VAR CONSTANT 		
	MAX_SEND_STRING_SIZE									:	INT := 1024;
END_VAR
VAR_OUTPUT CONSTANT
{attribute 'displaymode':='binary'}
	OPTION_SYSLOG_WITH_FACILITY_SEVERITY_CODE				:	BYTE := 2#0000_0001;
{attribute 'displaymode':='binary'}
	OPTION_SYSLOG_WITH_RFC_HEADER							:	BYTE := 2#0000_0010;
{attribute 'displaymode':='binary'}
	OPTION_SYSLOG_WITH_CR									:	BYTE := 2#0000_0100; 
	{attribute 'displaymode':='binary'}
	OPTION_SYSLOG_WITH_LF									:	BYTE := 2#0000_1000; 
{attribute 'displaymode':='binary'}
//	OPTION_SYSLOG_WITH_TCP_MODE								:	BYTE := 2#0001_0000;
{attribute 'displaymode':='binary'}
	OPTION_SEND_STORED_MSG_WITH_DISABLE						: 	BYTE := 2#0010_0000; //Send stored messages if FB gets disabled to clear buffer
{attribute 'displaymode':='binary'}
	OPTION_ENABLE_BUFFER_ERROR								: 	BYTE := 2#0100_0000; //The FB changes to error state if the buffer was not emptied in time 	
{attribute 'displaymode':='binary'}
	OPTION_ENABLE_DEBUG										:	BYTE := 2#1000_0000; //Creates ADS log entries for conection events and errors
END_VAR
VAR_INPUT
	Enable													: 	BOOL;	//Enables sending new messages
	ResetTrig												:	BOOL;	//Ack error message
{attribute 'displaymode':='binary'}
	Options													:	BYTE := OPTION_SYSLOG_WITH_FACILITY_SEVERITY_CODE ; //option constants are alreay predefined, so they can accordingly be passed symbolically to the block
	SizeOfBuffer											:	UDINT := 2560; //Size of memory allocated from ads router memory pool by DoubleBuffer instance
	LocalHost	 											: 	T_IPv4Addr;  	//Local (client) address. String containing an (Ipv4) Internet Protocol dotted address. 
	LocalPort												:	UDINT := 515;	//Local (client) Internet Protocol (IP) port. (TCP Port = 1468) *)	
	RemoteHost	 											: 	T_IPv4Addr;  	//Remote (server) address. String containing an (Ipv4) Internet Protocol dotted address. 
	RemotePort												:	UDINT := 514;	//Remote (server) Internet Protocol (IP) port. (TCP Port = 1468) 
	Facility												:	BYTE := 16; 	//Default local 16
	Severity 												:	BYTE := 7; 		//0=Emergency/1=Alert/2=Critical/3=Error/4=Warning/5=Notice/6=Informational/7=Debug
	Tag														:	STRING(32) := ''; //Process name or local host by default
	LogPriorityLevel										:	UINT := 0; 		//Correlate to EventClass prioritys - see Para.EVENT_HANDLING_CONFIG prioritys
END_VAR                 				
VAR_OUTPUT              				        			
	Online													:	BOOL;		//TRUE if coonection is sucessful etablished
	hSocket													: 	T_HSOCKET ; //UDP Socket handle
	CntNoOfStoredMsgs										:	INT;
	TimeSendMsgs											:	TIME;
	Busy													: 	BOOL;  //Sending busy
	Error													: 	BOOL;	//Error occured
{attribute 'displaymode':='hex'}
	ErrorId													:	UDINT;	//See Beckhoff TF6310/ADS documentation for more information regarding error code
	ErrorFnc												:	STRING(20); //Error source 
	WinsockErrorId											:	E_WinsockError; //Winsocket error enum - see TF6310 documentation for further information
END_VAR
VAR
(* Memory ************************************************************)
	State													: 	INT := 0;
	StartTimeSendMsgs										:	TIME;
	SendErrorCnt											:	UINT;
	HeaderString											:	STRING;
	SendString												:	STRING(MAX_SEND_STRING_SIZE);
	SendStringLen											:	INT;
	_Severity												:	BYTE;
	LastMessageData											: 	LogbookData;
	LastEventClass											:	E_TcEventClass := TC2_SYSTEM.TCEVENTCLASS_NONE;
	
(* Trigger *****************************************************************)

(* Timer ******************************************************************)

(* Blocks ***************************************************************)
	DblBuffer												:	DoubleBuffer;
	SocketClose												:	FB_SocketClose := (tTimeout := DEFAULT_ADS_TIMEOUT);
	SocketUdpCreate 										:	FB_SocketUdpCreate := (tTimeout := DEFAULT_ADS_TIMEOUT);
	SocketUdpSend											:	FB_SocketUdpSendTo := (tTimeout := T#10S);

(* Dummys *******************************************************************)
	i,j														:	INT;
END_VAR
(* 
Facality Description:
00 Kernel message
01 user-level messages
02 mail system
03 system daemons
04 security/authorization messages
05 messages generated internally by syslogd
06 line printer subsystem
07 network news subsystem
08 UUCP subsystem
09 clock daemon
10 security/authorization messages
11 FTP daemon
12 NTP subsystem
13 log audit
14 log alert
15 clock daemon
16 local10
17 local11
18 local12
19 local13
20 local14
21 local15
22 local16
23 local17

Severity Description:
0 Emergency
1 Alert
2 Critical
3 Error
4 Warning
5 Notice
6 Informational
7 Debug
*)

(* Logbook subscriber to send sys log messages via UDP 				*)
(********************************************************************)

(* Server connection ************************************************)
	CASE state OF
	0:
		IF Error
		THEN
			IF NOT Enable OR ResetTrig 
			THEN //Reset error
				Error										:= FALSE;
				ErrorId										:= 0;
				ErrorFnc									:= '';	
				WinsockErrorId								:= WSOK;			
			END_IF		
		ELSIF Online
		THEN
			IF DblBuffer.ReadyToRead 			
			THEN
				CntNoOfStoredMsgs							:= 0;
				StartTimeSendMsgs							:= TIME();

				SocketUdpSend(
					sSrvNetId	:= , 
					hSocket		:= hSocket, 
					sRemoteHost	:= RemoteHost, 
					nRemotePort	:= RemotePort, 
					cbLen		:= DblBuffer.SizeOfDataToRead, 
					pSrc		:= DblBuffer.pDataToRead, 
					bExecute	:= TRUE, 
					tTimeout	:= , 
					bBusy		=> , 
					bError		=> , 
					nErrId		=> );
													
				state										:= 20;
			END_IF
		ELSIF Enable			
		THEN
			DblBuffer.SizeOfMemory							:= SizeOfBuffer;
			SocketUdpCreate(bExecute := FALSE);
			SocketClose(bExecute := FALSE);
			SocketUdpSend(bExecute := FALSE);
			Online											:= FALSE;
			Busy											:= TRUE;
			Error											:= FALSE;
			ErrorId											:= 0;
			ErrorFnc										:= '';	
			WinsockErrorId									:= WSOK;
			
			IF NOT SocketUdpCreate.bBusy
				AND NOT SocketClose.bBusy
				AND NOT SocketUdpSend.bBusy
			THEN
				state										:= 10;
			END_IF	
		ELSE //Disabled
			IF NOT DblBuffer.Empty AND Options.5
			THEN //Write rest of buffer
				IF NOT DblBuffer.ReadyToRead THEN DblBuffer.setReadyToRead(TRUE); END_IF 
				CntNoOfStoredMsgs							:= 0;
				StartTimeSendMsgs							:= TIME();
				SocketUdpSend(
					sSrvNetId	:= , 
					hSocket		:= hSocket, 
					sRemoteHost	:= RemoteHost, 
					nRemotePort	:= RemotePort, 
					cbLen		:= DblBuffer.SizeOfDataToRead, 
					pSrc		:= DblBuffer.pDataToRead, 
					bExecute	:= TRUE, 
					tTimeout	:= , 
					bBusy		=> , 
					bError		=> , 
					nErrId		=> );
				State										:= 20;
			ELSE //Close socket
				State										:= 30;
			END_IF			
		END_IF

	(* Create Socket *******************************************************)
	10: 
		SocketUdpCreate(
			sSrvNetId	:= , 
			sLocalHost	:= LocalHost, 
			nLocalPort	:= LocalPort, 
			bExecute	:= TRUE, 
			tTimeout	:= , 
			bBusy		=> , 
			bError		=> , 
			nErrId		=> , 
			hSocket		=> hSocket);
			
		IF NOT SocketUdpCreate.bBusy
		THEN
			IF SocketUdpCreate.bError
			THEN
				Error										:= TRUE;
				ErrorId										:= SocketUdpCreate.nErrId;
				ErrorFnc									:= 'SocketUdpCreate';
				WinsockErrorId								:= ADSERROR_TO_WSERROR(ErrorId);
				
				IF (Options AND OPTION_ENABLE_DEBUG) = 1
				THEN
					AdsLogError(CONCAT('LogbookClientSysLog | SocketUdpCreate %s | error id 16#', DWORD_TO_HEXSTR(TO_DWORD(ErrorID),4,FALSE)) ,HSOCKET_TO_STRING(SocketUdpCreate.hSocket));
				END_IF	

				state										:= 30;
			ELSE				
				hSocket.remoteAddr.sAddr					:= RemoteHost;
				hSocket.remoteAddr.nPort					:= RemotePort;
				
				IF (Options AND OPTION_ENABLE_DEBUG) = 1
				THEN
					AdsLogError(CONCAT('LogbookClientSysLog | SocketUdpCreate %s done', '') , HSOCKET_TO_STRING(SocketUdpCreate.hSocket));
				END_IF	
				
				Online 										:= TRUE;
				state										:= 0;
			END_IF		
			SocketUdpCreate(bExecute:= FALSE);
		END_IF		
		
	(* Send message ****************************************************)
	20:
		SocketUdpSend(
			sSrvNetId	:= , 
			hSocket		:= hSocket, 
			sRemoteHost	:= RemoteHost, 
			nRemotePort	:= RemotePort, 
			cbLen		:= DblBuffer.SizeOfDataToRead, 
			pSrc		:= DblBuffer.pDataToRead, 
			bExecute	:= TRUE, 
			tTimeout	:= , 
			bBusy		=> , 
			bError		=> , 
			nErrId		=> );
					
		IF NOT SocketUdpSend.bBusy
		THEN
			IF SocketUdpSend.bError
			THEN
				IF SendErrorCnt >= 3
				THEN
					Error									:= TRUE;
					ErrorId									:= SocketUdpSend.nErrId;
					ErrorFnc								:= 'SocketUdpSend';
					WinsockErrorId							:= ADSERROR_TO_WSERROR(ErrorId);
	
					IF (Options AND OPTION_ENABLE_DEBUG) = 1
					THEN
						AdsLogError(CONCAT('LogbookClientSysLog | SocketUdpSend %s | error id 16#', DWORD_TO_HEXSTR(TO_DWORD(ErrorID),4,FALSE)) ,HSOCKET_TO_STRING(SocketUdpCreate.hSocket));
					END_IF	
					
					State									:= 30; //Close socket
				ELSE //Try to send a second time
					SendErrorCnt							:= SendErrorCnt + 1;
				END_IF
			ELSE				
				SendErrorCnt								:= 0;	
				State										:= 0;			
			END_IF 
			DblBuffer.setReadyToRead(FALSE);
			SocketUdpSend(bExecute := FALSE);
		END_IF
		
	(* Close socket ***********************************************)
	30:	
		SocketClose(
			sSrvNetId	:= , 
			hSocket		:= SocketUdpCreate.hSocket, 
			bExecute	:= TRUE, 
			tTimeout	:= , 
			bBusy		=> , 
			bError		=> , 
			nErrId		=> );

		IF NOT SocketClose.bBusy
		THEN
			Online											:= FALSE;
			IF SocketClose.bError 
				AND NOT Error
			THEN
				Error										:= TRUE;
				ErrorId										:= SocketClose.nErrId;
				ErrorFnc									:= 'SocketUdpClose';
				WinsockErrorId								:= ADSERROR_TO_WSERROR(ErrorId);
				
				IF (Options AND OPTION_ENABLE_DEBUG) = 1
				THEN
					AdsLogError( CONCAT('LogbookClientSysLog | SocketClose %s | error id 16#', DWORD_TO_HEXSTR(TO_DWORD(ErrorID),4,FALSE)) ,HSOCKET_TO_STRING(SocketClose.hSocket));
				END_IF

				state										:= 0;				
			ELSE    
				IF (Options AND OPTION_ENABLE_DEBUG) = 1
				THEN
					AdsLogError( CONCAT('LogbookClientSysLog | SocketClose %s done', '') , HSOCKET_TO_STRING(SocketClose.hSocket));
				END_IF	
                                        
				state										:= 0;
			END_IF		
			SocketClose(bExecute := FALSE);
		END_IF		
			
	END_CASE
	
(* Status *****************************************************************)
	Busy 													:= State <> 0;
	
(**************************************************************************)

METHOD PUBLIC FINAL addNewMessage : BOOL //Return value = TRUE if execution successful finished
VAR_IN_OUT
	data													:	LogbookData;
END_VAR
	IF Enable AND NOT Error
	THEN	
		LastMessageData									:= Data;
		LastEventClass.0								:= LastMessageData.Options.8;
		LastEventClass.1								:= LastMessageData.Options.9;
		LastEventClass.2								:= LastMessageData.Options.10;
		LastEventClass.3								:= LastMessageData.Options.11;
		
		CASE LastEventClass OF
		TC2_SYSTEM.TCEVENTCLASS_NONE		: _Severity		:= Severity; 		
		TC2_SYSTEM.TCEVENTCLASS_MESSAGE		: _Severity		:= 4;				
		TC2_SYSTEM.TCEVENTCLASS_HINT		: _Severity		:= 5;				
		TC2_SYSTEM.TCEVENTCLASS_STATEINFO	: _Severity		:= 6;				
		TC2_SYSTEM.TCEVENTCLASS_INSTRUCTION	: _Severity		:= 6;			 											
		TC2_SYSTEM.TCEVENTCLASS_WARNING		: _Severity		:= 4;	 			
		TC2_SYSTEM.TCEVENTCLASS_MAINTENANCE	: _Severity		:= 1;	 				 														
		TC2_SYSTEM.TCEVENTCLASS_ALARM		: _Severity		:= 0;	 			
		TC2_SYSTEM.TCEVENTCLASS_PARAMERROR	: _Severity		:= 3;	 			
		ELSE                                                                                     
			_Severity									:= 7;				
		END_CASE
	
		IF (LogPriorityLevel = 0 OR_ELSE GetEventClassPriority(LastEventClass) > LogPriorityLevel)
			AND_THEN CreateMsg(LastMessageData.Msg,LastMessageData.Timestamp ,_Severity)
		THEN
			IF DblBuffer.addData(ADR(SendString),TO_UDINT(SendStringLen)) <> S_OK
				AND Options.6
			THEN
				Error										:= TRUE;
				ErrorId										:= HRESULT_TO_ADSERROR(DblBuffer.hr);	
			ELSE
				CntNoOfStoredMsgs							:= CntNoOfStoredMsgs + 1;
			END_IF
		END_IF
		
		addNewMessage										:= NOT Error;	
	ELSE
		addNewMessage										:= FALSE;	
	END_IF
END_METHOD

METHOD PRIVATE FINAL createMsg : BOOL
VAR_IN_OUT
	MsgTxt													:	T_MaxString; (* 80/255 Zeichen *)
	MsgTime													:	TIMESTRUCT;	
	Severity												:	BYTE;
END_VAR                 									
VAR                     									
	TimeStamp												:	STRING(20);
	LenTxt													:	UDINT;
	LenHeader												:	UDINT;
END_VAR
	//Create Syslog msg
	IF (Options AND OPTION_SYSLOG_WITH_FACILITY_SEVERITY_CODE) <> 0 
	THEN 
		HeaderString 										:= REPLACE('<P>',BYTE_TO_STRING(SHL(FACILITY,3) OR (Severity AND BYTE#0000_0111)),1,2);
		             										
	ELSE             										
		HeaderString 										:= '';
	END_IF
	
	IF (Options AND OPTION_SYSLOG_WITH_RFC_HEADER) <> 0 
	THEN 
		//Sep 10 08:31:10
		CASE MsgTime.wMonth OF
		1: HeaderString 									:= CONCAT(HeaderString, ' Jan ');
		2: HeaderString 									:= CONCAT(HeaderString, ' Feb ');
		3: HeaderString 									:= CONCAT(HeaderString, ' Mar ');
		4: HeaderString 									:= CONCAT(HeaderString, ' Apr ');
		5: HeaderString 									:= CONCAT(HeaderString, ' May ');
		6: HeaderString 									:= CONCAT(HeaderString, ' Jun ');
		7: HeaderString 									:= CONCAT(HeaderString, ' Jul ');
		8: HeaderString 									:= CONCAT(HeaderString, ' Aug ');
		9: HeaderString 									:= CONCAT(HeaderString, ' Seb ');
		10:HeaderString 									:= CONCAT(HeaderString, ' Oct ');
		11:HeaderString 									:= CONCAT(HeaderString, ' Nov ');
		12:HeaderString 									:= CONCAT(HeaderString, ' Dec ');
		END_CASE
			
		HeaderString 										:= CONCAT(HeaderString,WORD_TO_STRING(MsgTime.wDay));
		HeaderString 										:= CONCAT(HeaderString, ' ');
					
		IF MsgTime.wHour <10 
		THEN
			TimeStamp 										:= CONCAT(' 0',WORD_TO_STRING(MsgTime.wHour));
		ELSE
			TimeStamp 										:= WORD_TO_STRING(MsgTime.wHour);
		END_IF
		
		TimeStamp 											:= CONCAT(TimeStamp,':');
		
		IF MsgTime.wMinute < 10 
		THEN
			TimeStamp 										:= CONCAT(TimeStamp,CONCAT('0',WORD_TO_STRING(MsgTime.wMinute)));
		ELSE          										
			TimeStamp 										:= CONCAT(TimeStamp,WORD_TO_STRING(MsgTime.wMinute));
		END_IF
		
		TimeStamp 											:= CONCAT(TimeStamp,':');
		
		IF MsgTime.wSecond < 10 
		THEN
			TimeStamp 										:= CONCAT(TimeStamp,CONCAT('0',WORD_TO_STRING(MsgTime.wSecond)));
		ELSE
			TimeStamp 										:= CONCAT(TimeStamp,WORD_TO_STRING(MsgTime.wSecond));
		END_IF
		HeaderString 										:= CONCAT(HeaderString,TimeStamp);
		HeaderString 										:= CONCAT(HeaderString,' ');
					
		(* ' sourcename eintragen (IP) *)
		HeaderString 										:= CONCAT(HeaderString, hSocket.localAddr.sAddr ); 
		HeaderString 										:= CONCAT(HeaderString,' '); 
		
		(* Tag *)
		IF Len(Tag) > 0
		THEN
			HeaderString									:= CONCAT(HeaderString,Tag);
			HeaderString 									:= CONCAT(HeaderString,' '); 
		END_IF
	END_IF
	
	IF Options.2 
	THEN //CR
		MsgTxt												:= CONCAT(MsgTxt,'$r');
	END_IF
	
	IF Options.3 
	THEN //LF
		MsgTxt												:= CONCAT(MsgTxt,'$n');
	END_IF
	
	(* Msg *)
	SendString												:= HeaderString;
	SendStringLen											:= MIN(MAX_SEND_STRING_SIZE,(LEN(HeaderString) + Len(MsgTxt)));
	MEMCPY(ADR(SendString) + LEN(HeaderString), ADR(MsgTxt) , INT_TO_UDINT(LEn(MsgTxt)));
	SendString[SendStringLen] 								:= 0; //Terminate string
	
	CreateMsg												:= TRUE;
END_METHOD

PROPERTY PUBLIC optAdd_CR : BOOL
GET
optAdd_CR := Options.2;
END_GET
SET
OPtions.2 := optAdd_CR;
END_SET
END_PROPERTY

PROPERTY PUBLIC optAdd_LF : BOOL
GET
optAdd_LF := Options.3;
END_GET
SET
Options.3 := optAdd_LF;
END_SET
END_PROPERTY

PROPERTY PUBLIC optEnabelDebugMode : BOOL
GET
optEnabelDebugMode := Options.7;
END_GET
SET
Options.7 := optEnabelDebugMode;
END_SET
END_PROPERTY

PROPERTY PUBLIC optEnableBufferError : BOOL
GET
optEnableBufferError := Options.6;
END_GET
SET
OPtions.6				:= optEnableBufferError;
END_SET
END_PROPERTY

PROPERTY PUBLIC optEnableFacilitySeverityCode : BOOL
GET
 optEnableFacilitySeverityCode := Options.0;
END_GET
SET
Options.0 := optEnableFacilitySeverityCode;
END_SET
END_PROPERTY

PROPERTY PUBLIC optEnableRFCHeader : BOOL
GET
optEnableRFCHeader := Options.1;
END_GET
SET
Options.1 := optEnableRFCHeader;
END_SET
END_PROPERTY

PROPERTY PUBLIC optSendMsgIfDisabled : BOOL
GET
optSendMsgIfDisabled := Options.5;
END_GET
SET
Options.5 := optSendMsgIfDisabled;
END_SET
END_PROPERTY

{attribute 'monitoring' := 'call'}
PROPERTY PUBLIC isBusy : BOOL
GET
isBusy											:= DblBuffer.Full and Enable and not Error and DblBuffer.fillLevel >= MAX_BUFFER_LEVEL;
END_GET
END_PROPERTY

END_FUNCTION_BLOCK

// POUs/Logging/LogbookSubWriteFile
{attribute 'no_check' := ''}
//The LogbooSubWriteFile writes log entries handover by the LogbookPuplisher into txt files
//The files could be stored or overwritten on a daily (Today/Yesterday), weekly (1-7 days) or monthly base (1-31 days) - see DeleteMode Parameter  
{attribute 'enable_dynamic_creation'}
FUNCTION_BLOCK LogbookSubWriteFile IMPLEMENTS I_LogbookSubscriber
VAR CONSTANT
	MAX_BUFFER_LEVEL										:	INT := 85; //If buffer fill level reaches 85% Fb will appear as "busy2 to the LogBookPuplisher 
END_VAR
VAR_OUTPUT CONSTANT 
	STRING_LINE_END_SIGN									: STRING(6) := PARAM.LOGBOOK_SUB_WRT_FILE_LINE_END_SIGN; //e.g. $n
	DELAY_CLOSE_FILE										: TIME := PARAM.LOGBOOK_SUB_WRT_FILE_DELAY_FILE_CLOSE;  //see library parameter to customize parameter	
		
	DELETE_MODE_DAILY										: INT := 0; //FB will write a file with <Filename>_TODAY and rename existing file to <Filename>_YESTERDAY on a new day
	DELETE_MODE_WEEKLY										: INT := 1; //FB will create a file for each day of week <Filenme>_DAY_1..7
	DELETE_MODE_MONTHLY										: INT := 2; //FB will create a file for each day of month <Filenme>_DAY_n (n=1..31) 
	DELETE_MODE_DISABLED									: INT := 3; //FB will write an endless file, see options .7 to start with an empty file on a new day  

	{attribute 'displaymode':='binary'}
	OPTION_ADD_TIMESTAMP_TO_MSG								: BYTE := 2#0000_0001; //Add message time to file entry - see next option for date option
	{attribute 'displaymode':='binary'}
	OPTION_ADD_DATE_TO_TIMESTAMP							: BYTE := 2#0000_0010; //Only active if option "OPTION_ADD_TIMESTAMP_TO_MSG" is set 
	{attribute 'displaymode':='binary'}
	OPTION_ADD_CLASS_TO_MSG									: BYTE := 2#0000_0100; //Event class text will be added to entries
	{attribute 'displaymode':='binary'}
	OPTION_ENABLE_BUFFER_ERROR								: BYTE := 2#0100_0000; //The FB changes to error state if the buffer was not emptied in time 
	{attribute 'displaymode':='binary'}
	OPTION_START_WITH_NEW_FILE								: BYTE := 2#1000_0000; //Create empty file with enable flag instead open and continie existing file
END_VAR                     								
VAR_INPUT                   								
	Enable													: BOOL; //Enable write log entries to file
	ResetTrig												: BOOL; //Reset internal error 
{attribute 'displaymode':='binary'}
	Options													: BYTE := 2#00000000; // Bit 0 = Add msg timestamp to entry string 	
	DeleteMode												: INT(DELETE_MODE_DAILY..DELETE_MODE_DISABLED) := DELETE_MODE_DAILY;
	Path													: STRING := 'C:\temp'; //Path and filename
	Filetype												: STRING(6) := '.log'; //file tpye
	LoggedDay												: WORD;	//Init for logged day of month to avoid new and empty log file after reboot.
	SizeOfBuffer											: UDINT := 2560; //Size of memory allocated from router pool to accumulate messages until they get written to the file (0=Write message immediately)
END_VAR                     								
VAR_IN_OUT                  								
	SystemTime												: TIMESTRUCT; //System time
END_VAR                     								
VAR_OUTPUT       
	CntNoOfStoredMsgs										: INT; //No of messages added to buffer 

	hFile													: UINT;  
	Busy													: BOOL; //Write msg to file active   
	Error													: BOOL;        			
{attribute 'displaymode':='hex'}					
	ErrorId													: UDINT; //Ads error Id of file handling function blocks
END_VAR                     								
VAR            
//local ************************************************************************************
	State													: INT := 0;
	LastLoggedDay											: WORD;
	Rebooted												: BOOL;
	LastMessageData											: LogbookData;
	StartTimeWriteData										: TIME;	
	TimeWriteFile											: TIME; 
	MemMessage												: U_MAX_STRING;
	MemLenStrEndLine										: INT;	
	MemStartOfEndLine										: DINT;	
	MemPath													: STRING;
	
//trigger *********************************************************************************

//timer ***********************************************************************************
	tonCloseFile											:	ton;

//instances ***********************************************************************************     
	DblBuffer												: DoubleBuffer;        								
	FILEOPEN												: FB_FileOpen := (sNetId:='',tTimeout:=DEFAULT_ADS_TIMEOUT, ePath:=PATH_GENERIC);
	FILECLOSE												: FB_FileClose := (sNetId:='',tTimeout:=DEFAULT_ADS_TIMEOUT);
	FILEWRITE												: FB_FileWrite := (sNetId:='',tTimeout:=DEFAULT_ADS_TIMEOUT);
	FILEDELETE												: FB_FileDelete := (sNetId:='',tTimeout:=DEFAULT_ADS_TIMEOUT);
	FILERENAME												: FB_FileRename := (sNetId:='',tTimeout:=DEFAULT_ADS_TIMEOUT, ePath:=PATH_GENERIC);

//Dummys ****************************************************************************************
	i,j,n													: INT;
	_UINT													:	UINT;
END_VAR

	(* Logbook subscriber write messages to file			*)
	(********************************************************)

(* Sequence started by method "NewMessage" or a new day ***************************************************)
	CASE State OF
	0:	
		IF Error
		THEN
			IF ResetTrig OR NOT Enable
			THEN
				Error										:= FALSE;
				ErrorId										:= 0;
				FileOpen(bExecute:=FALSE);
				FileClose(bExecute:=FALSE);
				FileDelete(bExecute:=FALSE);
				FileRename(bExecute:=FALSE);
				FileWrite(bExecute:=FALSE);
			END_IF
		ELSIF Enable
		THEN
			IF SystemTime.wDay = 0
			THEN
				Error										:= TRUE;
				ErrorId										:= E_AdsErr.DEVICE_INVALIDPARM; //Systemtime invalid 				
			ELSIF hFile = 0 // close last before opening next file
				AND(LastLoggedDay <> SystemTime.wDay OR MemPath <> Path) 			
			THEN //create new or overwrite existing file if new day begins
				DblBuffer.SizeOfMemory						:= SizeOfBuffer;
						
				MemLenStrEndLine							:= LEN(STRING_LINE_END_SIGN);
				MemStartOfEndLine							:= TO_DINT(LIMIT(1,PARAM.LOGBOOK_MAX_MSG_STRING_LENGHT - TO_UDINT(MemLenStrEndLine) + 1, PARAM.LOGBOOK_MAX_MSG_STRING_LENGHT - 1));
				Rebooted									:= LastLoggedDay = 0;
 	
				(* Init last logged day of month and path on startup *)
				IF Rebooted 
				THEN 
					MemPath  								:= Path;
					LastLoggedDay 							:= SEL(LoggedDay > 0, 0, LoggedDay); 
				END_IF	
				
				CASE DeleteMode OF
				DELETE_MODE_WEEKLY: //Day 1 to 7
					FileOpen.sPathName 						:= CONCAT(Path, CONCAT('_DAY_',WORD_TO_STRING(SystemTime.wDayOfWeek)));
					CASE SystemTime.wDayOfWeek OF
					0:FileOpen.sPathName 					:= CONCAT(FileOpen.sPathName,'_SUN' );
					1:FileOpen.sPathName 					:= CONCAT(FileOpen.sPathName,'_MON' );
					2:FileOpen.sPathName					:= CONCAT(FileOpen.sPathName,'_TUE' );
					3:FileOpen.sPathName 					:= CONCAT(FileOpen.sPathName,'_WED' );
					4:FileOpen.sPathName 					:= CONCAT(FileOpen.sPathName,'_THU' );
					5:FileOpen.sPathName 					:= CONCAT(FileOpen.sPathName,'_FRI' );
					6:FileOpen.sPathName 					:= CONCAT(FileOpen.sPathName,'_SAT' );
					ELSE
						FileOpen.sPathName 					:= CONCAT(FileOpen.sPathName,'_UNKNOW' );
					END_CASE
					
				DELETE_MODE_MONTHLY: //Every Month - Day 1-n
					FileOpen.sPathName 						:= CONCAT(Path, CONCAT('_',WORD_TO_STRING(SystemTime.wDay)));
					
				DELETE_MODE_DISABLED:		
					FileOpen.sPathName			 			:= Path;
					
				ELSE //DELETE_MODE_DAILY as default
					FileOpen.sPathName 						:= CONCAT(Path, '_TODAY');	//Today and yesterday
				
				END_CASE
				FileOpen.sPathName							:= CONCAT(FileOpen.sPathName,Filetype);
									
				IF DeleteMode <> DELETE_MODE_DISABLED AND LastLoggedDay <> SystemTime.wDay 
				THEN //New day - start with new file	
					FileOpen(bExecute:=FALSE,nMode := FOPEN_MODEWRITE OR FOPEN_MODETEXT OR FOPEN_MODEPLUS);							
					IF DeleteMode = DELETE_MODE_DAILY
					THEN //Rename old file first		
						FILERENAME(bExecute:=FALSE, sOldName := FileOpen.sPathName, sNewName := CONCAT(Path, CONCAT('_YESTERDAY',Filetype)));
						FILEDELETE(bExecute:=FALSE, sPathName := FILERENAME.sNewName );
						FileClose(bExecute:=hFile <> 0 , hFile := hFile);
						state								:= 10;
					ELSE //Create new file directly
						FileOpen(bExecute:=TRUE,nMode := FOPEN_MODEWRITE OR FOPEN_MODETEXT OR FOPEN_MODEPLUS);
						state								:= 1;
					END_IF
				ELSE //write endless file with given name and open existing one if selected 														
					FileOpen(bExecute:= TRUE , nMode:=SEL(Options.7 ,FOPEN_MODEAPPEND,FOPEN_MODEWRITE) OR FOPEN_MODETEXT OR FOPEN_MODEPLUS );
					state									:= 1;
				END_IF	 	
	
				(* Record current day of detected new beginning day *)
				LastLoggedDay 								:= SystemTime.wDay;	
				MemPath  									:= Path;
				
			ELSE
				tonCloseFile(IN := NOT DblBuffer.Empty ,PT := DELAY_CLOSE_FILE); 
				IF DblBuffer.ReadyToRead
					OR tonCloseFile.Q
				THEN
					IF NOT DblBuffer.ReadyToRead THEN DblBuffer.setReadyToRead(TRUE); END_IF 
					FILEWRITE.pWriteBuff 					:= DblBuffer.pDataToRead;
					FILEWRITE.cbWriteLen 					:= DblBuffer.SizeOfDataToRead;
					FILEWRITE.bExecute						:= DblBuffer.SizeOfDataToRead > 0; //Set Write file as marker

					FileClose.bExecute						:= SystemTime.wDay > 0
																AND(LastLoggedDay <> SystemTime.wDay OR MemPath <> Path)
																AND hFile <> 0
																OR tonCloseFile.Q; //Set close file as marker
																
					tonCloseFile(IN := FALSE); //Reset timer....
					CntNoOfStoredMsgs						:= 0;
					StartTimeWriteData						:= TIME();
					
					IF hFile = 0
					THEN
						FileOpen(bExecute:= TRUE , nMode:=SEL(Options.7 ,FOPEN_MODEAPPEND,FOPEN_MODEWRITE) OR FOPEN_MODETEXT OR FOPEN_MODEPLUS ); //Reopen file first
						State								:= 1;
					ELSE
						FILEWRITE(hFile := hFile); //Start write file for efficiency 		
						State								:= 2;
					END_IF					
				END_IF			
			END_IF
						
		ELSE //Not enabled
			IF NOT DblBuffer.Empty
			THEN //Write rest of buffer
				IF NOT DblBuffer.ReadyToRead THEN DblBuffer.setReadyToRead(TRUE); END_IF 
				FILEWRITE(bExecute:=TRUE,hFile:= hFile , pWriteBuff := DblBuffer.pDataToRead, cbWriteLen := DblBuffer.SizeOfDataToRead);	
				CntNoOfStoredMsgs							:= 0;
				StartTimeWriteData							:= TIME();
				FileClose.bExecute							:= TRUE;  //Close file after writing
				State										:= SEL(hFile <> 0 , 1, 2) ; //Open file if not opened
			ELSIF hFile <> 0
			THEN
				FileClose(bExecute:=TRUE , hFile := hFile);
				state										:= 3;	
			END_IF
        END_IF
     
	(* Open file *******************************************************************************)                                          	
	1:                       	
		FileOpen();                                     	
		IF NOT FileOpen.bBusy                           	
		THEN                                            	
			IF FileOpen.bError                          	
			THEN            
				Error										:= TRUE;                            	
				ErrorId										:= FileOpen.nErrId;
				State										:= 0;
			ELSE                                     	
				hFile										:= FileOpen.hFile;       	
				State										:= SEL(FILEWRITE.bExecute, 0, 2) ;
			END_IF
			FileOpen(bExecute:=FALSE);			
		END_IF

	(* Write data to file **********************************************************************)
	2: 
		FILEWRITE(hFile:= hFile);	
		IF NOT FILEWRITE.bBusy
		THEN
			
			IF FILEWRITE.bError
			THEN
				Error										:= TRUE;       
				ErrorId										:= FILEWRITE.nErrId;
				state										:= 0;
			ELSE  
				State										:= SEL(FileClose.bExecute, 0, 3);	
			END_IF		
			TimeWriteFile									:= TIME() - StartTimeWriteData;		
			DblBuffer.setReadyToRead(FALSE);	
			FILEWRITE(bExecute:=FALSE);   	
		END_IF

	(* Close File ******************************************************************************)
	3: 
		FileClose(hFile:= hFile);
		IF NOT FileClose.bBusy
		THEN
			IF FileClose.bError
			THEN
				Error										:= TRUE;       
				ErrorId										:= FileClose.nErrId;
				State										:= 0;
			ELSE                                        	
				hFile										:= 0;
				State										:= 0;
			END_IF
			FileClose(bExecute:=FALSE);
		END_IF

	(* Delete old file and rename exisiting file ********************************************************) 
	10: 
		FileClose();
		FileDelete(bExecute:=NOT FileClose.bBusy);
		IF NOT FileDelete.bBusy AND NOT FileClose.bBusy
		THEN
			IF FileDelete.bError
			THEN //No issue, maybe file is not existing
			//	Error										:= TRUE;       
			//	ErrorId										:= FileDelete.nErrId;
				State										:= 11;
			ELSIF FileClose.bError
			THEN
			//	Error										:= TRUE;       
			//	ErrorId										:= FileClose.nErrId;
				State										:= 11;			
			ELSE                                        	
				State										:= 11;
			END_IF
			FileDelete(bExecute:=FALSE); FileClose(bExecute:=FALSE);
		END_IF
		
	11: //Rename last file to create a new and empty file for today
		FILERENAME(bExecute:=TRUE);
		IF NOT FILERENAME.bBusy
		THEN
			IF FILERENAME.bError
			THEN //No issue, maybe file does not exist
			//	Error										:= TRUE;       
			//	ErrorId										:= FILERENAME.nErrId;
				State										:= 1;
			ELSE                                        	
				State										:= 1;
			END_IF
			FILERENAME(bExecute:=FALSE);	
			FileOpen(bExecute:= TRUE); //Start create new file for today										
		END_IF		
	ELSE
		;
	END_CASE

(* Ack ErrorIds **********************************************************)
	Busy 													:= State <> 0;
(**************************************************************************)

METHOD PUBLIC FINAL addNewMessage : BOOL //Return value = TRUE if execution successful finished
VAR_IN_OUT
	data													:	LogbookData;
END_VAR
	IF Enable AND NOT Error
	THEN		
		CntNoOfStoredMsgs								:= CntNoOfStoredMsgs + 1;
		LastMessageData									:= Data;

		MEMSET(ADR(MemMessage),0,SIZEOF(MemMessage));
		IF Options.0 AND Options.1 //Add date and time to text
		THEN
			MemMessage.text								:=	SYSTEMTIME_TO_STRING(LastMessageData.Timestamp);						
			MemMessage.text 							:=	CONCAT(MemMessage.text, ';');

		ELSIF Options.0 //Add only msg timestamp to text		
		THEN
			MemMessage.text								:=	SYSTEMTIME_TO_STRING(LastMessageData.Timestamp);
			MemMessage.text								:=	MID(MemMessage.text, 12 , 12); //Cut out time
			MemMessage.text 							:=	CONCAT(MemMessage.text, ';');
		END_IF      

		IF Options.2 //Add class of message to text
		THEN
			_UINT.0 									:= LastMessageData.Options.8;
			_UINT.1 									:= LastMessageData.Options.9;
			_UINT.2 									:= LastMessageData.Options.10;
			_UINT.3 									:= LastMessageData.Options.11;		
			MemMessage.text								:= CONCAT(MemMessage.text, GetEventClassText(_UINT));	
			MemMessage.text 							:= CONCAT(MemMessage.text, ';');			
		END_IF
	
		MemMessage.text 								:= CONCAT(MemMessage.text, LastMessageData.Msg);

		IF LEN(MemMessage.text) < MemStartOfEndLine
		THEN //Still enough space for end line signs
			MemMessage.text 							:= CONCAT(MemMessage.text,STRING_LINE_END_SIGN );
		ELSE //Overwrite last chars with endline signs
			MEMCPY(ADR(MemMessage.text[MemStartOfEndLine]),ADR(STRING_LINE_END_SIGN),TO_UDINT(MemLenStrEndLine));
		END_IF
		
		IF DblBuffer.addString(MemMessage.text) <> S_OK
			AND Options.6
		THEN
			Error										:= TRUE;
			ErrorId										:= HRESULT_TO_ADSERROR(DblBuffer.hr);	
		END_IF
		
		addNewMessage									:= NOT Error;
	ELSE
		addNewMessage									:= FALSE;
	END_IF
END_METHOD

PROPERTY PUBLIC optAddDateToMsg : BOOL
GET
optAddDateToMsg := Options.1;
END_GET
SET
Options.1 := optAddDateToMsg and optAddTimeToMsg;
END_SET
END_PROPERTY

PROPERTY PUBLIC optAddEventClassToMsg : BOOL
GET
optAddEventClassToMsg := Options.2;
END_GET
SET
Options.2 := optAddEventClassToMsg ;
END_SET
END_PROPERTY

PROPERTY PUBLIC optAddTimeToMsg : BOOL
GET
optAddTimeToMsg := Options.0;
END_GET
SET
IF optAddTimeToMsg 
THEN
	Options.0 := TRUE;
ELSE
	Options.0 := Options.1 := FALSE;
END_IF
END_SET
END_PROPERTY

PROPERTY PUBLIC optEnableBufferError : BOOL
GET
optEnableBufferError := Options.6;
END_GET
SET
OPtions.6				:= optEnableBufferError;
END_SET
END_PROPERTY

PROPERTY PUBLIC optSendMsgIfDisabled : BOOL
GET
optSendMsgIfDisabled := Options.5;
END_GET
SET
Options.5 := optSendMsgIfDisabled;
END_SET
END_PROPERTY

PROPERTY PUBLIC optStartNewFile : BOOL
GET
optStartNewFile := Options.7;
END_GET
SET
OPtions.7				:= optStartNewFile;
END_SET
END_PROPERTY

{attribute 'monitoring' := 'call'}
PROPERTY PUBLIC isBusy : BOOL
GET
isBusy											:= DblBuffer.Full and Enable and not Error and DblBuffer.fillLevel >= MAX_BUFFER_LEVEL;
END_GET
END_PROPERTY

END_FUNCTION_BLOCK

// POUs/Motion/TF50xx-NC/00_Base/AxFbBase
//Axis FB template, inherited Execute, Busy etc from FbBase   
FUNCTION_BLOCK AxFbBase EXTENDS FbBase 
VAR_INPUT
	rAxis													: REFERENCE TO AXIS_REF := 0; //Reference to AXIS_REF 
END_VAR
VAR_IN_OUT
END_VAR
VAR_OUTPUT
	Active													: BOOL ; // If the axis movement is controlled by several functions, the Active output of each block indicates that the axis executes the command. 
	CmdAborted												: BOOL ; // TRUE if a command is interrupted through another block (Busy and Error = FALSE)
	ErrorText												: STRING(40); //Error text with name of internal used FB which causes the error
END_VAR
VAR 
	LastErrorId												: UDINT := 0; //Last error id
END_VAR

END_FUNCTION_BLOCK

// POUs/Motion/TF50xx-NC/00_Base/I_AxNcBase
INTERFACE I_AxNcBase EXTENDS __SYSTEM.IQueryInterface

METHOD PUBLIC noAction : BOOL //Return value = TRUE if busy of home and motion 
VAR_INPUT
END_VAR
END_METHOD

{attribute 'monitoring' := 'call'}
PROPERTY rAdmin : REFERENCE TO AxAdmin
GET
END_GET
END_PROPERTY

{attribute 'monitoring' := 'call'}
PROPERTY rAxisRef : REFERENCE TO AXIS_REF
GET
END_GET
END_PROPERTY

{attribute 'monitoring' := 'call'}
PROPERTY rErrHdl : REFERENCE to ERROR_HDL
GET
END_GET
SET
END_SET
END_PROPERTY

METHOD reset : Bool
VAR_INPUT
END_VAR
END_METHOD

{attribute 'monitoring' := 'call'}
PROPERTY rHome : REFERENCE TO AxHoming
GET
END_GET
END_PROPERTY

{attribute 'monitoring' := 'call'}
PROPERTY rPara : REFERENCE TO AxPara
GET
END_GET
END_PROPERTY

END_INTERFACE

// POUs/Motion/TF50xx-NC/01_Main/AxAdmin
{attribute 'no_check'}
//Nc-axis administration - Axis reset, set operation and override
//based on Tc2_MC2 library
//Call cyclic to update AXIS_REF.status
FUNCTION_BLOCK AxAdmin 
VAR_INPUT
	ResetTrig												:	BOOL := FALSE; // Reset NC Error and restart current cmd if possible
	Enable													: 	BOOL := FALSE; // Cyclic NCAxis enable operational - FALSE = Stop 
	EnablePos												: 	BOOL := FALSE; // feed enable positiv 
	EnableNeg												: 	BOOL := FALSE; // feed enable negative 
	BufferMode												:	MC_BufferMode := MC_Aborting;	(* 	MC_Aborting,
																									MC_Buffered,
																									MC_BlendingLow,
																									MC_BlendingPrevious,
																									MC_BlendingNext,
																									MC_BlendingHigh *) 
                                							
	Override												:	LREAL; // Override 
	PT_Ready												:	TIME := T#10MS; //Delay of ready signal after NC-Axis has been enabled
	ShowNCErrIfDisabled										:	BOOL := FALSE; // FB reports and NC-Error even if axis has been diabled
	EnableNcDebugFlag										:	BOOL := FALSE; //TRUE writes every MC2 start command into TwinCAT and Windows logger. 
	ExeMcStopToDisable										:	BOOL := FALSE; //Initiats the execution of MC_Stop on a running axis if "Enable" is set to FALSE
	Dec														:	LREAL := 0.0; //Deceleration during disable, if the value is 0, the deceleration parameterized with the last Move command is used / see also ExeMcStopToDisable
	Jerk													:	LREAL := 0.0; //Jerk during disable, if the value is 0, the deceleration parameterized with the last Move command is used / see also ExeMcStopToDisable
	rAxis													:	REFERENCE TO AXIS_REF := 0;

END_VAR                         							
VAR_IN_OUT                      							
END_VAR                         							
VAR_OUTPUT                      							
	EnableOK												:	BOOL; // Enable is send to NC
	Ready													:	BOOL; // NC-Axis is enabled
	StartRel												:	BOOL; // NC-Axis is enabled (Ready) and in PTPMode, not protected or motion command disabeld and at least one movment direction enabled
	Busy													:	BOOL; //Internal MC functionblock is busy
//	Done													:	BOOL; 
	Error													:	BOOL; // Error occured at one internal MC functionblock 
{attribute 'displaymode':='hex'}
	ErrorID													:	UDINT;// ErrorID of one internal MC functionblock 
	ErrorText												:	STRING(40); // Name of internal MC functionblock which has an error
END_VAR
VAR
(* Cache **************************************************************************)
	MethSeqEnable											: 	BOOL := TRUE;	(* NCAchse BTB/Freigabe setzen - FALSE = Stop, auch ueber Methoden set/reset bar *)
	                        	
(* Timer *)                 	
	TON_Ready												:	TON;

(* Trigger *)

(* Instanzierung der MC Bausteine *******************************************************)
	MC_Power												: MC_Power;
	MC_Reset												: MC_Reset;
	MC_Stop													: MC_Stop;
	MC_ReadDriveAddress										: MC_ReadDriveAddress;
	
(* Dummy Speicher **********************************************************)

END_VAR

	(*	NC axis administration															*)
	(*	Call function-block cyclic to enable axis and refresh AxisRef.Status structure	*)
	(************************************************************************************)

(* abortinf function-block-call if reference is invalid *********************************)
IF NOT __ISVALIDREF(rAxis) THEN
	EnableOK												:= FALSE;
	Busy													:= NOT Error;
	Ready													:= FALSE;
	Error													:= TRUE;
	ErrorId													:= E_adsErr.DEVICE_INVALIDPARM;
//	Done													:= FALSE;
	StartRel												:= FALSE;
	ErrorText												:= 'Reference rAxis invalid (0)';
	RETURN;	
END_IF

(* reading axis-status from NCtoPLC-channel ***********************************************)
	rAxis.ReadStatus();
	raxis.PlcToNc.ControlDWord.31							:= EnableNcDebugFlag;
	
(* read drive address information **********************************************)
IF MC_ReadDriveAddress.DriveAddress.SlaveAddress = 0
	OR MC_ReadDriveAddress.Busy
THEN
	MC_ReadDriveAddress(
		Axis:= rAxis, 
		Execute:= NOT rAxis.Status.DriveDeviceError AND NOT rAxis.Status.IoDataInvalid AND(NOT ResetTrig OR NOT MC_ReadDriveAddress.Error), 
		Done=> , 
		Busy=> , 
		Error=> , 
		ErrorID=> , 
		DriveAddress=> );
END_IF

(* Enable OK ****************************************************************************)
	EnableOK 												:= Enable AND MethSeqEnable;

(* stop **********************************************************************************)
	MC_Stop(
		Axis		:= rAxis, 
		Execute		:= rAxis.Status.Moving AND NOT EnableOK AND ExeMcStopToDisable, 
		Deceleration:= Dec, 
		Jerk		:= Jerk, 
		Options		:= , 
		Done		=> , 
		Busy		=> , 
		Active		=> , 
		CommandAborted=> , 
		Error		=> , 
		ErrorID		=> );

(* set axis operational  *****************************************************************)
	MC_Power(
		Enable			:= 	EnableOK 
							OR 
							MC_Power.Active AND MC_Stop.Busy,
		Enable_Positive	:= EnablePos,
		Enable_Negative	:= EnableNeg,
		Override		:= Override,
		BufferMode		:= (* PwrBufferMode *),
		Axis			:= rAxis,
		Status			=> ,
		Busy			=> ,
		Active			=> ,
		Error			=> ,
		ErrorID			=> );

(* Reset axis ****************************************************************)
	MC_Reset(
		Execute	:= 	ResetTrig 
					AND (NOT rAxis.Status.ProtectedMode OR rAxis.Status.DriveDeviceError)
					AND (rAxis.NcToPlc.ErrorCode <> 0 OR NOT rAxis.Status.HasJob)
					OR MC_Reset.Execute,
		Axis	:= rAxis,
	//	Done	=> Done,
		Busy	=> ,
		Error	=> ,
		ErrorID	=> );
		
	MC_Reset.Execute										:= FALSE; 	

(********************************************************************************)
(* axis status																	*)
(********************************************************************************)
	(* Delay axis is ready to move *)
	TON_Ready(
		IN := MC_Power.Status,//ControlLoopClosed
		PT 	:= PT_Ready, 
		Q	=> Ready);

	(* Axis Ready to Start *)
	StartRel												:= Ready
																AND rAxis.Status.PTPmode
																AND NOT rAxis.Status.ProtectedMode
																AND NOT rAxis.Status.MotionCommandsLocked
																AND (MC_Power.Enable_Negative OR MC_Power.Enable_Positive);
                                							
(********************************************************************************)
(* Ctrl Status 															 		*)
(********************************************************************************)
	Busy													:= (MC_Power.Busy AND NOT MC_Power.Status) //Show MC_Power busy only if as long as axis is not enabled  
																OR MC_Stop.Busy 
																OR MC_Reset.Busy;
	IF NOT ShowNCErrIfDisabled AND NOT EnableOK
	THEN
		Error												:= FALSE;
		ErrorId												:= 0;
		ErrorText											:= '';	
	ELSIF MC_Power.Error
		AND NOT MC_Reset.Execute
	THEN
		Error												:= TRUE;
		ErrorId												:= MC_Power.ErrorID;
		ErrorText											:= CONCAT('MC_Power ErrorId: ', UDINT_TO_STRING(Errorid));
	ELSIF MC_Reset.Execute  								
		AND MC_Reset.Error  								
	THEN                    								
		Error												:= TRUE;
		ErrorId												:= MC_Reset.ErrorID;
		ErrorText											:= CONCAT('MC_Reset ErrorId: ', UDINT_TO_STRING(Errorid));
	ELSIF MC_Stop.Execute  								
		AND MC_Stop.Error  								
	THEN                    								
		Error												:= TRUE;
		ErrorId												:= MC_Stop.ErrorID;
		ErrorText											:= CONCAT('MC_Stop ErrorId: ', UDINT_TO_STRING(Errorid));
	ELSIF rAxis.NcToPlc.ErrorCode <> 0 
	THEN
		Error												:= TRUE;
		ErrorId												:= rAxis.NcToPlc.ErrorCode;
		ErrorText											:= CONCAT('NC ErrorId: ', UDINT_TO_STRING(Errorid));
	ELSIF MC_ReadDriveAddress.Execute  								
		AND MC_ReadDriveAddress.Error  								
	THEN                    								
		Error												:= TRUE;
		ErrorId												:= MC_ReadDriveAddress.ErrorID;
		ErrorText											:= CONCAT('MC_ReadDriveAddress ErrorId: ', UDINT_TO_STRING(Errorid));
		
	ELSE                    								
		Error												:= FALSE;
		ErrorId												:= 0;
		ErrorText											:= '';
	END_IF

(**************************************************************************************************)

METHOD PUBLIC forceFeed : BOOL //Return value = TRUE if execution finished 
VAR_INPUT
	IN														:	booL;
END_VAR
THIS^.EnableNeg 											:= IN;
THIS^.EnablePos 											:= IN;

forceFeed 													:=  TRUE;
END_METHOD

PROPERTY PUBLIC isResetting : BOOL
GET
isResetting := MC_Reset.Busy;
END_GET
END_PROPERTY

PROPERTY PUBLIC isStopping : BOOL
GET
isStopping := MC_Stop.Busy;
END_GET
END_PROPERTY

METHOD PUBLIC reset : BOOL //Return value = True if Busy
//required parameter
//rAxis
VAR_INPUT
	IN						:	BOOL; //Force to send a reset, even if the axis is not in error state. With FALSE, reset will be only send if axis has an error
END_VAR
IF NOT __ISVALIDREF(rAxis) 
THEN
	Busy													:= NOT Error;
	Error													:= TRUE;
	ErrorId													:= E_AdsErr.DEVICE_INVALIDPARM;
//	Done													:= FALSE;
	ErrorText												:= 'Reference rAxis invalid (0)';
	RETURN;             								
END_IF

	MC_Reset(
		Execute	:= NOT rAxis.Status.ProtectedMode
					AND (	ResetTrig 
							OR IN 
							OR rAxis.NcToPlc.ErrorCode <> 0 
							OR NOT rAxis.Status.HasJob) ,
		Axis	:= rAxis,
		Done	=> ,
		Busy	=> Busy,
		Error	=> Error,
		ErrorID	=> ErrorId);

	IF Error 
	THEN
		ErrorText											:= SEL(MC_Reset.Error , '' ,  CONCAT('Error MC_Reset id: ',  UDINT_TO_STRING(Errorid)));
	ELSE            										
		ErrorText											:= '';
	END_IF          										
	                	
	reset													:= Busy;
END_METHOD

METHOD PUBLIC seqEnable : BOOL //Return = Ready - Enable and disabel per method from external
VAR_INPUT
	IN														:	BOOL;
END_VAR
THIS^.MethSeqEnable 										:= IN;
seqEnable													:= Ready;
END_METHOD

END_FUNCTION_BLOCK

// POUs/Motion/TF50xx-NC/01_Main/AxHoming
{attribute 'no_check'}
//Nc-axis homing control 
//based on Tc2_MC2 library
//Call cyclic to send calibration cam signal to NC even if homing is not running 
FUNCTION_BLOCK AxHoming EXTENDS AxFbBase
VAR_OUTPUT CONSTANT
	FNC_HALT												:	INT := 0;
	FNC_HOMING												:	INT := 1;
	FNC_SETPOS												:	INT := 2;
END_VAR                     								
VAR_INPUT                   								
	Fnc														:	INT (FNC_HALT..FNC_SETPOS):= FNC_HALT;
	BufferMode												:	MC_BufferMode := MC_Aborting;(* 	MC_Aborting,
																												MC_Buffered,
																											MC_BlendingLow,
																											MC_BlendingPrevious,
																											MC_BlendingNext,
																											MC_BlendingHigh *)
	Mode													:	MC_HomingMode := MC_DefaultHoming; (*	MC_DefaultHoming 		default homing as defined in the SystemManager encoder parameters
																						MC_Direct	 			static Homing forcing position from user reference  								
																						MC_ForceCalibration	set the calibration flag without perfoming any motion OR changing the position
																						MC_ResetCalibration	resets the calibration flag without perfoming any motion OR changing the position *)
	AcceptBlockedDrive										:	BOOL := TRUE; 	(* AcceptBlockedDrive *)
	CalibrationCam											:	BOOL := FALSE;
	Pos														:	LREAL := DEFAULT_HOME_POSITION;
	SetPosModeRel 											: 	BOOL := FALSE;	(* RELATIVE=True, ABSOLUTE=False (Default) *)
	SetPosOptions 											: 	ST_SetPositionOptions;                            					
END_VAR                     								
VAR_IN_OUT                  	
END_VAR                     	
VAR_OUTPUT                  	
END_VAR
VAR
(* Zwischenspeicher **************************************************************************)
	MemFnc													:	INT := -1;
	MemFncAct												:	INT := -1;
	MCFctTxt												:	STRING(25);
	BusyIntern												:	BOOL := FALSE;
                            								
(* Timer *)                 								
                            								
(* Trigger *)               	
	rtExecuteMethod											:	R_TRIG;

(* Instanzierung der MC Bausteine *******************************************************)
	MC_Home													: 	MC_Home;
	MC_Halt													: 	MC_Halt;
	MC_SetPosition											:	MC_SetPosition;

END_VAR

	(* Axis homing control																*)
	(************************************************************************************)

(* Cyclic ****************************************************************************************)
	Cyclic();

(* Execute ***************************************************************************************)
	rtExecute(CLK := Execute);
	IF rtExecute.Q AND NOT rtExecuteMethod.Q
(*		AND MemFnc < 0 neue Fnc immer zulassen weil alter gleichzeitig zurueckgesetzt werden *)
	THEN
		MemFnc 												:= Fnc ;
		Busy												:= TRUE;
		Done												:= FALSE;
		Active												:= FALSE;
		Error												:= FALSE;
		ErrorID												:= 0;
		CmdAborted											:= FALSE;
		ErrorText											:= '';
	END_IF
	
(* Call Method ***********************************************************************************)
	CASE MemFnc OF
	FNC_HALT												:	Halt(Execute);
	FNC_HOMING												:	Homing(Execute);
	FNC_SETPOS												:	SetPos(Execute);
	-1:                                     				
		IF NOT rtExecute.CLK                   				
		THEN                                				
			Busy											:= FALSE;
			Done											:= FALSE;
			Error											:= FALSE;
			ErrorID											:= 0;
			Active											:= FALSE;
			CmdAborted										:= FALSE;
			ErrorText										:= '';
		END_IF
	ELSE
		Busy												:= FALSE;
		Done												:= FALSE;
		Active												:= FALSE;
		Error												:= Execute;
		ErrorID												:= E_AdsErr.DEVICE_INVALIDPARM;
		CmdAborted											:= FALSE;
		ErrorText											:= CONCAT('invalid parameter value(s) Fnc no: ' , INT_TO_STRING(MemFnc));
	END_CASE

(*************************************************************************************************)

METHOD PRIVATE _MCIntern : BOOL
VAR_INPUT
END_VAR
	(* Internal MC Action														*)
	(***************************************************************)

(* Check Pointer **********************************************************************)
IF NOT __ISVALIDREF(rAxis) THEN
	Done													:= FALSE;
	Busy													:= NOT Error;
	Active													:= FALSE;
	CmdAborted												:= FALSE;
	Error													:= TRUE;
	ErrorId													:= E_AdsErr.DEVICE_INVALIDPARM;
	ErrorText												:= 'Reference rAxis invalid (0)';
	MemFnc													:= SEL(Execute , -1 ,MemFnc); 
	RETURN;
END_IF

(* flag Execute ***********************************************************************)
	rtExecuteMethod(CLK := Execute OR rtExecute.Q);
	IF rtExecuteMethod.Q
	THEN
		MC_Home.Execute										:= FALSE;
		MC_Halt.Execute										:=	FALSE;
		MC_SetPosition.Execute								:= FALSE;
		BusyIntern											:= FALSE;
		MemFncAct 											:= MemFnc;
	END_IF

(* ctrl programm ******************************************************************************)
	CASE MemFncAct OF
	FNC_HALT:
		MC_Halt.Execute										:=	Execute; (* Execute if axis is not locked *)
		MC_Halt.BufferMode									:= MC_Aborting (* BufferMode *);
		MC_Halt.Deceleration 								:= 0.0;
		MC_Halt.Jerk 										:= 0.0;

	FNC_HOMING:
		IF (Execute OR MC_Halt.Busy) (* new cmd or stop last cmd busy *)
			AND NOT rAxis.NcToPlc.StateDWord.2  (* NotMoving *)
			AND NOT MC_Home.Busy and not Mc_Home.Done
			AND NOT rAxis.NcToPlc.StateDWord.5 (* Protected *) (* not if axis coupled or in NCI group *)
			AND NOT MC_Halt.Error AND NOT MC_Halt.CommandAborted
		THEN
			MC_Halt.Execute									:=	TRUE;
			MC_Halt.BufferMode								:= MC_Aborting;
			BusyIntern										:= TRUE;
		ELSE
			MC_Home.Execute									:= Execute OR MC_Halt.Execute AND BusyIntern;
			MC_Home.Position								:= Pos;
			MC_Home.HomingMode								:= Mode;
			MC_Home.BufferMode								:= MC_Aborting;
			MC_Home.Options.ClearPositionLag				:= TRUE;
			MC_Halt.Execute									:=	FALSE;
			BusyIntern										:= FALSE;
		END_IF

	FNC_SETPOS:
		MC_SetPosition.Execute								:= Execute;
		MC_SetPosition.Position								:= Pos;
		MC_SetPosition.Mode									:= SetPosModeRel;
		MC_SetPosition.Options								:= SetPosOptions;

	ELSE
		Error												:= TRUE;
		ErrorId												:= E_AdsErr.DEVICE_INVALIDPARM;
		ErrorText											:= CONCAT('invalid parameter value(s) - Fnc no ', INT_TO_STRING(MemFncAct)) ;
	END_CASE

(******************************************************************************)
(* Work MC Blocks 																				*)
(******************************************************************************)

	(* Halt/Stop *)
	MC_Halt(Axis:= rAxis);

	(* Referenzieren *)
	MC_Home(Axis:= rAxis, bCalibrationCam := CalibrationCam);

	(* Set Position *)
	MC_SetPosition(Axis	:= rAxis);

(******************************************************************************)
(* Ctrl Status 																					*)
(******************************************************************************)
	IF MemFncAct = FNC_HALT
	THEN
		MCFctTxt											:= 'MC_HALT';
		Done 												:= MC_Halt.Done;
		Busy 												:= MC_Halt.Busy;
		Active 												:= MC_Halt.Active;
		CmdAborted 	 										:= MC_Halt.CommandAborted;
		Error												:=	MC_Halt.Error;
		ErrorId												:= MC_Halt.ErrorId;
		ErrorText											:= SEL(Error , '' ,  CONCAT('Error MC_HALT id: ',  UDINT_TO_STRING(Errorid)));

	ELSIF BusyIntern
	THEN
		MCFctTxt											:= CONCAT('BUSY INTERN at Fnc no: ', INT_TO_STRING(MemFncAct));
		Busy												:= BusyIntern;
		Done 												:= FALSE;
		Active 												:= FALSE;
		CmdAborted 											:= FALSE;
		Error												:=	FALSE;
		ErrorId												:= 0;
		ErrorText											:= '';

	ELSIF MemFncAct = FNC_HOMING
	THEN
		MCFctTxt											:= 'MC_Home';
		Done 												:= MC_Home.Done;
		Busy 												:= MC_Home.Busy;
		Active 												:= MC_Home.Active;
		CmdAborted 	 										:= MC_Home.CommandAborted;
		Error												:=	MC_Home.Error;
		ErrorId												:= MC_Home.ErrorId;
		ErrorText											:= SEL(Error , '' ,  CONCAT('Error MC_Home id: ',  UDINT_TO_STRING(Errorid)));

	ELSIF MemFncAct = FNC_SETPOS
	THEN
		MCFctTxt											:= 'MC_SetPosition';
		Done 												:= MC_SetPosition.Done;
		Busy 												:= MC_SetPosition.Busy;
		Active 												:= Busy;
		CmdAborted 	 										:= FALSE;
		Error												:=	MC_SetPosition.Error;
		ErrorId												:= MC_SetPosition.ErrorId;
		ErrorText											:= SEL(Error , '' ,  CONCAT('Error MC_SetPosition id: ',  UDINT_TO_STRING(Errorid)));

	ELSE
		MCFctTxt											:= SEL(BusyIntern, 'NoAction' , 'Busy intern');
		Busy												:= BusyIntern;
		Done 												:= FALSE;
		Active 												:= FALSE;
		CmdAborted 											:= FALSE;
		IF Error THEN LastErrorId := ErrorId; END_IF
		Error												:=	FALSE;
		ErrorId												:= 0;
		ErrorText											:= '';
	END_IF


(* End funcktion *********************************************************************************)
	IF 	NOT rtExecuteMethod.CLK 
		AND NOT Busy 
		AND NOT Error 
		AND NOT Done 
		AND NOT Active 
		AND NOT CmdAborted
	THEN
		IF MC_SetPosition.Busy
			OR MC_Halt.Busy
			OR MC_Home.Busy
		THEN (* Ablauffehler , es darf kein Baustein an dieser Stelle Busy sein *)
			MemFnc											:= -2;
		ELSE                								
			MemFnc											:= -1;
		END_IF
	END_IF

(* Return value ***********************************************************************************)
	_MCIntern												:= TRUE;
	
(**************************************************************************************************)
END_METHOD

METHOD PRIVATE cyclic : BOOL
//required parameter
//rAxis
VAR_INPUT
END_VAR
IF NOT __ISVALIDREF(rAxis) 
THEN
	Done													:= FALSE;
	Busy													:= NOT Error;
	Active													:= FALSE;
	CmdAborted												:= FALSE;
	Error													:= TRUE;
	ErrorId													:= E_AdsErr.DEVICE_INVALIDPARM;
	ErrorText												:= 'Reference rAxis invalid (0)';
	RETURN;
END_IF

(* accept setvalue-barrier (e.g. hardware limit switch) ********************************)
	rAxis.PlcToNc.AxisModeDWord.8 							:= AcceptBlockedDrive;

(* Send Calibration Cam cylic to the nc ************************************************)
	rAxis.PlcToNc.ControlDWord.5							:= CalibrationCam;

(***************************************************************************************)
	cyclic													:= TRUE;
	
(***************************************************************************************)
END_METHOD

METHOD PUBLIC halt : BOOL //Return value = TRUE if busy
//required parameter
//rAxis
VAR_INPUT
	Execute													:	BOOL;
END_VAR
MemFnc				 										:= FNC_HALT;
THIS^.Execute												:= Execute;
_MCIntern();            									
halt 														:= Busy;
END_METHOD

METHOD PUBLIC homing : BOOL //Return value = TRUE if busy
//required parameter
//rAxis
//Pos
//HomingMode
//BufferMode
VAR_INPUT
	Execute													:	BOOL;
END_VAR
MemFnc 														:= FNC_HOMING;
THIS^.Execute												:= Execute;
_MCIntern();            									
Homing														:= Busy;
END_METHOD

METHOD PUBLIC setPos : BOOL //Return value = TRUE if busy
//required parameter
//rAxis
//Pos
//SetPosModeRel
//SetPosOptions
VAR_INPUT
	Execute													:	BOOL;
END_VAR
MemFnc														:= FNC_SETPOS;
THIS^.Execute												:= Execute;
_MCIntern();            									
SetPos														:= Busy;
END_METHOD

END_FUNCTION_BLOCK

// POUs/Motion/TF50xx-NC/02_Options/Parameter/AxPara
{attribute 'no_check'}
//FB to read and write NC axis parameter. 
//The FB can be enherided and derivatived methods of SeqRead/SeqWrite used for application specific parameter.
//The extended methods need to call the super class at the beginning and return true if execution will be finished. The allowed states for new parameter are 1..99
FUNCTION_BLOCK AxPara EXTENDS AxRWParaBase
VAR_OUTPUT CONSTANT
END_VAR                                 					
VAR_INPUT                               					                                   	                                        	
	AxisID													: 	UDINT;				(* ID der Achse *)

	(* zu schreibende Achparameter *)
	SetLimitPosActive										: 	BOOL;
	SetLimitNegActive										:	BOOL;
	SetLimitPos												: 	LREAL;
	SetLimitNeg												: 	LREAL;
                                    						
	SetRefFlag												:	BOOL;
                                    						
	SetTargetPosWindow										:	LREAL;
	SetTargetPosWindowMonitoring							:	BOOL;
	SetPosRangeWindow										: 	LREAL;
	SetPosRangeWindowMonitoring								:	BOOL;

	SetDynamicsRefVelocity									: 	LREAL;
	SetDynamicsMaxVelocity									: 	LREAL;
	SetG0Velocity											: 	LREAL;
	SetRefVelocityPos										: 	LREAL;
	SetRefVelocityNeg										: 	LREAL;
	SetManVelocityFast										: 	LREAL;
	SetManVelocitySlow										: 	LREAL;

	SetKv													: 	LREAL;
	SetJerk													: 	LREAL;
	SetAcc													: 	LREAL;
	SetDec													: 	LREAL;
	SetMaxPosLagValue										: 	LREAL;
	SetMaxPosLagFilterTime									: 	LREAL;
	
	SetMaxPosLagMonitoring									: 	BOOL;
                                        					
	SetModuloFactor 										:	LREAL;
	SetToleranceWindowModuloStart							:	LREAL;
	SetInvertEncCoutingDir									:	BOOL; //UINT;
                                        					
	SetEncScalingNumerator									:	LREAL; //Scaling idx 16#6 replaced by Numerator and Denominator
	SetEncScalingDenominator								:	LREAL; //Scaling idx 16#6 replaced by Numerator and Denominator
	SetPosBias												: 	LREAL; (* NC positon offset *)
	SetReferenceSystem										:	UDINT; //incremental, absolute, abs modulo
	SetCalibrationValue										: 	LREAL;	(* read/write only allowed for certain encoder types *)
	SetCalibrationMode										:	UDINT; 
	SetCalibrInvertDirForCamSearch							:	BOOL; (* TRUE=Cam search direction negative , read/write only allowed for certain encoder types *)
	SetCalibrInvertDirForSyncImpSearch						:	BOOL; (* TRUE=Sync impuls (off cam) search direction negative, read/write only allowed for certain encoder types *)
	
	SetInvertMotorPolarity									: 	BOOL; //UINT;
                                							  	
	SetBreakingDistancePos									: 	LREAL;
	SetBreakingDistanceNeg									: 	LREAL;
END_VAR                                 					
VAR_OUTPUT                              										
	Name													: STRING(30) := '';
	AxisType												: UDINT := 0; (* Nc axis type :
																								0	NOT DEFINED
																								1	Continuous axis (stepper motor)
																								2	Diskrete Achse (Eil/Schleich)
																								3	Continuous axis (stepper motor)
																								5	Encoder axis/ simulation axis *)
                                        					
	ChannelType												: UDINT := 1;(*  NC channel type:
																								1	Stantard,
																								2	Interpreter (CNC)
																								3	FIFO 
																								4	Kinematic *) 
                                        					
	EncType													: UDINT := 0;(* Encoder type:
																								0  	NOT DEFINED 
																								1  	Simulation Encoder (Incremental) 
																								2 	M3000 Encoder (Multi/Single-Turn) (Absolute) 
																								3 	M31x0 / M2000 Encoder (Incremental) 
																								4 	MDP 511 Encoder: EL7041, EL7342, EL5101, EL5151, EL2521, EL5021, IP5101 (Incremental) 
																								5	MDP 500/501 Enc.: EL5001, IP5009, KL5001 (SSI) (Absolute) 
																								6 	MDP 510 Encoder: KL5051, KL2502-30K Encoder (BiSSI)	(Incremental) 
																								7 	KL30xx Encoder (Analog) (Absolute) 
																								8 	SERCOS and EtherCAT SoE (Position)(Incremental) 
																								9 	SERCOS and EtherCAT SoE (Position and velocity) (Incremental) 
																								10 	Binary encoder (0/1)	(Incremental) 
																								11 	M2510 Encoder (Absolute) 
																								12 	FOX50 Encoder (Absolute) 
																								14 	AX2000 (Lightbus)(Incremental) 
																								15 	Provi-Drive MC (Simodrive 611U) (Incremental) 
																								16 	Universal encoder (variable bit mask) (Incremental) 
																								17 	NC back plane (Incremental) 
																								18 	Special CANopen type (e.g. Lenze Drive 9300) (Incremental) 
																								19	MDP 513 (DS402): CANopen and EtherCAT CoE (AX2xx-B1x0/B510, EL7201) (Incremental) 
																								20 	AX2xx-B900 (Ethernet) (Incremental) 
																								21 	KL5151 Encoder (Incremental) 
																								24 	IP5209 Encoder (Incremental) 
																								25 	KL2531/KL2541 Encoder (Stepper Motor) (Incremental) 
																								26 	KL2532/KL2542 Encoder (DC motor), KL2535/KL2545 (PWM current terminal) (Incremental) 
																								27 	Time base encoder (Time Base Generator) (Incremental) 
																								28 	TCom Encoder (Soft Drive) (Incremental) *)																				

	EncTypAbs												:	BOOL := 0; (* Encodertyp Abs = 1/ Rel = 0*)
	RefFlag													:	BOOL := 0; (* Axis is in reference *)
                                							
	LimitPosActive											: 	BOOL;
	LimitNegActive											:	BOOL;
	LimitPos												: 	LREAL;
	LimitNeg												: 	LREAL;

	TargetPosWindow											:	LREAL;
	TargetPosWindowMonitoring								:	BOOL;
	PosRangeWindow											: 	LREAL;
	PosRangeWindowMonitoring								:	BOOL;
                                							
	DynamicsRefVelocity										: 	LREAL;
	DynamicsMaxVelocity										: 	LREAL;
	G0Velocity												: 	LREAL;
	RefVelocityPos											: 	LREAL;
	RefVelocityNeg											: 	LREAL;
	ManVelocityFast											: 	LREAL;
	ManVelocitySlow											: 	LREAL;
                                							  	
	Kv														: 	LREAL;
	Jerk													: 	LREAL;
	Acc														: 	LREAL;
	Dec														: 	LREAL;
	MaxPosLagValue											: 	LREAL;
	MaxPosLagFilterTime										: 	LREAL;
	MaxPosLagMonitoring										: 	BOOL;
                                                              	
	InvertEncCoutingDir										: 	BOOL;
	ModuloFactor											: 	LREAL;
	ToleranceWindowModuloStart								: 	LREAL;
	EncScalingNumerator										:	LREAL;
	EncScalingDenominator									:	LREAL;
	EncScaling												: 	LREAL; //Factor of Numerator and Denominator
	PosBias													: 	LREAL;  (* Actual NC position offset *)
	ReferenceSystem											:	UDINT; //incremental, absolute
	CalibrationMode											:	UDINT;
	CalibrationValue										: 	LREAL;	(* read/write only allowed for certain encoder types  *)
	RefFlagDistance											: 	LREAL;	(* read/write only allowed for certain encoder types *)
	CalibrInvertDirForCamSearch								:	BOOL; (* TRUE=Cam search direction negative , read/write only allowed for certain encoder types *)
	CalibrInvertDirForSyncImpSearch							:	BOOL; (* TRUE=Sync impuls (off cam) search direction negative, read/write only allowed for certain encoder types *)

	InvertMotorPolarity										: 	BOOL;
                                							  	
	BreakingDistancePos										: 	LREAL;
	BreakingDistanceNeg										: 	LREAL;
	
END_VAR                         	


VAR
(* Zwischenspeicher ************************************************************)
	
(* Deklaration Trigger **********************************************************)

(* Zeiten ******************************************************************)

(* Bausteine ***************************************************************)
	ReadAdsPara												: ADSREAD := (NetId	:= '' , Port := AMSPORT_R0_NC, TmOut	:= DEFAULT_ADS_TIMEOUT);
	WriteAdsPara											: ADSWRITE := (NetId:= '' , Port := AMSPORT_R0_NC, TmOut	:= DEFAULT_ADS_TIMEOUT);

(* Dummy Speicher **********************************************************)

END_VAR

	(************************************************************************************)
	(*																					*)
	(*		B E C K H O F F   N E W   A U T O M A T I O N   T E C H N O L O G Y    		*)
	(*																					*)
	(*		Eiserstr.5	D-33415 Verl	Germany	phone:	+49-5246-0	www.Beckhoff.Com	*)
    (*																					*)
    (*		Bausteinbeschreibung	:	Read/Write axis parameter						*)
	(*		TwinCAT-Version			:	3.x or higher									*)
	(*																					*)
	(************************************************************************************)

(* Execute ***************************************************************************************)
	Super^();			
	
(*************************************************************************************************)

PROPERTY PROTECTED deviceAddrIsValid : BOOL
GET
deviceAddrIsValid := AxisId > 0;
END_GET
END_PROPERTY

METHOD PROTECTED getValue : BOOL //Return value = TRUE if execution finished and state incremented 
VAR_INPUT
	IDxGrp						:	UDINT;
	IDxOffs						:	UDINT;
	Len							:	UDINT;
	pActValue					:	PVOID; //Address of variable for actual value
	pSetValue					:	PVOID; //Address of variable for ser value variable, can be zero if no corresponding SetVariable exists
END_VAR

ReadAdsPara	(Read := TRUE, IDxGrp:=IDxGrp+AxisId, IDxOffs:=IDxOffs,LEN:=Len,DestAddr:=pActValue );
IF NOT ReadAdsPara.BUSY
THEN
	IF NOT ReadAdsPara.ERR 
	THEN 
		IF pSetValue <> 0 THEN MEMCPY(pSetValue, pActValue, Len); END_IF			
		state 												:= state + 1; 
	ELSE 		
		Busy												:= FALSE;
		Error												:= TRUE;
		ErrorId												:= ReadAdsPara.ERRID;
		ErrorText											:= CONCAT('Error read parameter in state:' , TO_STRING(state * -1));
		ErrorText											:= CONCAT(ErrorText , ' Id:');
		ErrorText											:= CONCAT(ErrorText , TO_STRING(ErrorId));
		State												:= 9999;
	END_IF	
	ReadAdsPara(Read := FALSE); 
	getValue												:= TRUE;									
END_IF
END_METHOD

METHOD PROTECTED seqRead : BOOL //Return value = TRUE if execution finished 
VAR_IN_OUT
	State							:	INT;
END_VAR
(* Execute read axis parameter ************************************)
	CASE state OF
	1..99: //read application spec parameter 
		seqRead												:= TRUE;
		
	1001: (* Name *************************************************************************************)
		IF LEN(Name) > 0 AND NOT ReadAdsPara.BUSY
		THEN
			state											:= state + 1;
		ELSE
			getValue(IDxGrp:= 16#4000,	IDxOffs := 16#2,	LEN := SIZEOF(Name),		pActValue := ADR(Name),			pSetValue := 0);
		END_IF

	1002: (* Axis Type ( Für Beschreibung Typen siehe AxPara) **********************************)
		IF AxisType <> 0 AND NOT ReadAdsPara.BUSY
		THEN
			state											:= state + 1;
		ELSE
			getValue(IDxGrp:= 16#4000,	IDxOffs := 16#3,	LEN := SIZEOF(AxisType),	pActValue := ADR(AxisType), 	pSetValue := 0);
		END_IF

	1003: (* NC Channel type ****************************************************************************************)
		IF ChannelType <> 0 AND NOT ReadAdsPara.BUSY
		THEN
			state											:= state + 1;
		ELSE
			getValue(IDxGrp:= 16#4000,	IDxOffs := 16#53,	LEN := SIZEOF(ChannelType),	pActValue := ADR(ChannelType), 	pSetValue := 0);
		END_IF

	1004: (* EncType ****************************************************************************************)
		IF EncType <> 0 AND NOT ReadAdsPara.BUSY
		THEN
			state											:= state + 1;
		ELSE
			getValue(IDxGrp:= 16#5000,	IDxOffs := 16#3,	LEN := SIZEOF(EncType),	pActValue := ADR(EncType), 		pSetValue := 0);
		END_IF
	
	1005: (* Endlagenlimit pos. ***********************************************************************)
		getValue(IDxGrp:= 16#5000,	IDxOffs := 16#E,	LEN := SIZEOF(LimitPos),	pActValue := ADR(LimitPos),  pSetValue := ADR(SetLimitPos) );	
	
	1006: (* Endlagenlimit neg ***********************************************************************)
		getValue(IDxGrp:= 16#5000,	IDxOffs := 16#D,	LEN := SIZEOF(LimitNeg),	pActValue := ADR(LimitNeg),  pSetValue := ADR(SetLimitNeg) );
		
	1007: (* Endlagenlimit pos aktiv ? ***************************************************************)
		IF getValue(IDxGrp:= 16#5000,	IDxOffs := 16#C,	LEN := SIZEOF(_UINT),	pActValue := ADR(_UINT),  pSetValue := 0)
		THEN
			SetLimitPosActive :=LimitPosActive				:= TO_BOOL(_UINT);
		END_IF

	1008: (* Endlagenlimit neg aktiv ? ***************************************************************)
		IF getValue(IDxGrp:= 16#5000,	IDxOffs := 16#B,	LEN := SIZEOF(_UINT),	pActValue := ADR(_UINT),  pSetValue := 0)
		THEN
			SetLimitNegActive :=LimitNegActive				:= TO_BOOL(_UINT);
		END_IF

	1009: (* Zielfenster ******************************************************************************)
		getValue(IDxGrp:= 16#4000,	IDxOffs := 16#16,	LEN := SIZEOF(TargetPosWindow),	pActValue := ADR(TargetPosWindow),  pSetValue := ADR(SetTargetPosWindow) );

	1010: (* Positionsfenster ************************************************************************)
		getValue(IDxGrp:= 16#4000,	IDxOffs := 16#10,	LEN := SIZEOF(PosRangeWindow),	pActValue := ADR(PosRangeWindow),  pSetValue := ADR(SetPosRangeWindow) );

	1011: (* Bezugsgeschwindigkeit (siehe Typenschild)*************************************)
		IF AxisType = 2 
		THEN
			state											:= state + 1;
		ELSE
			getValue(IDxGrp:= 16#7000,	IDxOffs := 16#101,	LEN := SIZEOF(DynamicsRefVelocity),	pActValue := ADR(DynamicsRefVelocity),  pSetValue := ADR(SetDynamicsRefVelocity) );
		END_IF
	
	1012: (* Max.Geschwindigkeit (ca. 90% der Bezugsgeschw.)***************************)
		IF AxisType = 2 
		THEN
			state											:= state + 1;
		ELSE
			getValue(IDxGrp:= 16#4000,	IDxOffs := 16#27,	LEN := SIZEOF(DynamicsMaxVelocity),	pActValue := ADR(DynamicsMaxVelocity),  pSetValue := ADR(SetDynamicsMaxVelocity) );
		END_IF
		
	1013: (* G0 Geschwindigkeit ****************************************************************)
		getValue(IDxGrp:= 16#4000,	IDxOffs := 16#A,	LEN := SIZEOF(G0Velocity),	pActValue := ADR(G0Velocity),  pSetValue := ADR(SetG0Velocity) );

	1014: (* Ref.Geschwindigkeit Pos **********************************************************)
		getValue(IDxGrp:= 16#4000,	IDxOffs := 16#6,	LEN := SIZEOF(RefVelocityPos),	pActValue := ADR(RefVelocityPos),  pSetValue := ADR(SetRefVelocityPos) );

	1015: (* Ref.Geschwindigkeit Neg **********************************************************)
		getValue(IDxGrp:= 16#4000,	IDxOffs := 16#7,	LEN := SIZEOF(RefVelocityNeg),	pActValue := ADR(RefVelocityNeg),  pSetValue := ADR(SetRefVelocityNeg) );

	1016: (* Man. Verfahrgeschwindigkeit fast *************************************************)
		getValue(IDxGrp:= 16#4000,	IDxOffs := 16#9,	LEN := SIZEOF(ManVelocityFast),	pActValue := ADR(ManVelocityFast),  pSetValue := ADR(SetManVelocityFast) );

	1017: (* Man. Verfahrgeschwindigkeit slow ***********************************************)
		getValue(IDxGrp:= 16#4000,	IDxOffs := 16#8,	LEN := SIZEOF(ManVelocitySlow),	pActValue := ADR(ManVelocitySlow),  pSetValue := ADR(SetManVelocitySlow) );

	1018: (* Kv ************************************************************************************)
		IF AxisType = 2
		THEN
			state											:= state + 1;
		ELSE
			getValue(IDxGrp:= 16#6000,	IDxOffs := 16#102,	LEN := SIZEOF(Kv),	pActValue := ADR(Kv),  pSetValue := ADR(SetKv) );
		END_IF

	1019: (* Ruck ************************************************************************************)
		IF AxisType = 2 
		THEN
			state											:= state + 1;
		ELSE
			getValue(IDxGrp:= 16#4000,	IDxOffs := 16#103,	LEN := SIZEOF(Jerk),	pActValue := ADR(Jerk),  pSetValue := ADR(SetJerk) );
		END_IF
		

	1020: (* Beschleunigung ***********************************************************************)
		IF AxisType = 2
		THEN
			state											:= state + 1;
		ELSE
			getValue(IDxGrp:= 16#4000,	IDxOffs := 16#101,	LEN := SIZEOF(Acc),	pActValue := ADR(Acc),  pSetValue := ADR(SetAcc) );
		END_IF

	1021: (* Verzoegerung ***************************************************************************)
		IF AxisType = 2 
		then
			state											:= state + 1;
		ELSE
			getValue(IDxGrp:= 16#4000,	IDxOffs := 16#102,	LEN := SIZEOF(Dec),	pActValue := ADR(Dec),  pSetValue := ADR(SetDec) );
		END_IF

	1022: (* Schleppabstand ***********************************************************************)	
		getValue(IDxGrp:= 16#6000,	IDxOffs := 16#12,	LEN := SIZEOF(MaxPosLagValue),	pActValue := ADR(MaxPosLagValue),  pSetValue := ADR(SetMaxPosLagValue) );

	1023: (* Skalierung ******************************************************************************)
		getValue(IDxGrp:= 16#5000,	IDxOffs := 16#6,	LEN := SIZEOF(EncScaling),	pActValue := ADR(EncScaling),  pSetValue := 0 );		

	1024: (* Positions Offset  ***********************************************************************)
		getValue(IDxGrp:= 16#5000,	IDxOffs := 16#7,	LEN := SIZEOF(PosBias),	pActValue := ADR(PosBias),  pSetValue := ADR(SetPosBias) );

	1025: (* Referenzposition (Nicht bei Absolut Encoder lesen)*******************************)
		IF EncType <> 2 AND EncType <> 5 AND EncType<> 7 AND EncType <> 11 AND EncType <> 12
		THEN
			getValue(IDxGrp:= 16#5000,	IDxOffs := 16#103,	LEN := SIZEOF(CalibrationValue),	pActValue := ADR(CalibrationValue),  pSetValue := ADR(SetCalibrationValue) );
		ELSE
			state											:= state +1;
		END_IF

	1026: (* Abstand Ref-Nocken Synchronimpuls (Nicht bei Absolut Encoder lesen) ****)
		IF EncType <> 2 AND EncType <> 5 AND EncType <> 7 AND EncType <> 11 AND EncType <> 12
		THEN
			getValue(IDxGrp:= 16#5100,	IDxOffs := 16#101,	LEN := SIZEOF(RefFlagDistance),	pActValue := ADR(RefFlagDistance),  pSetValue := 0 );
		ELSE
			state											:= state +1;
		END_IF

	1027: (* Drive direction **************************************************************)
		IF getValue(IDxGrp:= 16#7000,	IDxOffs := 16#6,	LEN := SIZEOF(_UINT),	pActValue := ADR(_UINT),  pSetValue := 0)
		THEN
			SetInvertMotorPolarity :=InvertMotorPolarity	:= TO_BOOL(_UINT);
			
		END_IF

	1028: (* Bremsweg positiv **********************************************************************)
		IF AxisType <> 2
		THEN
			state											:= state + 1;
		ELSE
			getValue(IDxGrp:= 16#4000,	IDxOffs := 16#303,	LEN := SIZEOF(BreakingDistancePos),	pActValue := ADR(BreakingDistancePos),  pSetValue := ADR(SetBreakingDistancePos ));
		END_IF

	1029: (* Bremsweg negativ *********************************************************************)
		IF AxisType <> 2 
		THEN
			state											:= state + 1;
		ELSE
			getValue(IDxGrp:= 16#4000,	IDxOffs := 16#304,	LEN := SIZEOF(BreakingDistanceNeg),	pActValue := ADR(BreakingDistanceNeg),  pSetValue := ADR(SetBreakingDistanceNeg ));

		END_IF

	1030: (* Schleppueberwachung Aktiv *********************************************************************)
		IF getValue(IDxGrp:= 16#6000,	IDxOffs := 16#10,	LEN := SIZEOF(_UINT),	pActValue := ADR(_UINT),  pSetValue := 0)
		THEN
			SetMaxPosLagMonitoring :=MaxPosLagMonitoring	:= TO_BOOL(_UINT);
			
		END_IF

	1031: (* Encodertyp Abs/Rel *********************************************************************)
		IF getValue(IDxGrp:= 16#5000,	IDxOffs := 16#1D,	LEN := SIZEOF(_UINT),	pActValue := ADR(_UINT),  pSetValue := 0)
		THEN
			EncTypAbs										:= TO_BOOL(_UINT);
			
		END_IF

	1032: (* Referenzierflag *********************************************************************)
		IF getValue(IDxGrp:= 16#5100,	IDxOffs := 16#9,	LEN := SIZEOF(_UINT),	pActValue := ADR(_UINT),  pSetValue := 0)
		THEN
			SetRefFlag :=RefFlag							:= TO_BOOL(_UINT);
		END_IF

	1033: (* Zielfenster Aktiv ******************************************************************)
		IF getValue(IDxGrp:= 16#4000,	IDxOffs := 16#15,	LEN := SIZEOF(_UINT),	pActValue := ADR(_UINT),  pSetValue := 0)
		THEN
			SetTargetPosWindowMonitoring :=TargetPosWindowMonitoring := TO_BOOL(_UINT);
			
		END_IF

	1034: (* Positionsfenster Aktiv ******************************************************************)
		IF getValue(IDxGrp:= 16#4000,	IDxOffs := 16#F,	LEN := SIZEOF(_UINT),	pActValue := ADR(_UINT),  pSetValue := 0)
		THEN
			SetPosRangeWindowMonitoring :=PosRangeWindowMonitoring := TO_BOOL(_UINT);
			
		END_IF

	1035: (* ModuloFaktor ******************************************************************)
		getValue(IDxGrp:= 16#5000,	IDxOffs := 16#9,	LEN := SIZEOF(ModuloFactor),	pActValue := ADR(ModuloFactor),  pSetValue := ADR(SetModuloFactor ));

	1036: (* Enc Zaehlrichtung ******************************************************************)
		IF getValue(IDxGrp:= 16#5000,	IDxOffs := 16#8,	LEN := SIZEOF(_UINT),	pActValue := ADR(_UINT),  pSetValue := 0)
		THEN
			SetInvertEncCoutingDir :=InvertEncCoutingDir := TO_BOOL(_UINT);
			
		END_IF

	1037: (* Toleranzfenster Modulo Start *******************************************************)
		getValue(IDxGrp:= 16#5000,	IDxOffs := 16#1B,	LEN := SIZEOF(ToleranceWindowModuloStart),	pActValue := ADR(ToleranceWindowModuloStart),  pSetValue := ADR(SetToleranceWindowModuloStart ));
		
	1038: (* Calibration cam search direction inverted *******************************************************)
		IF EncType <> 2 AND EncType <> 5 AND EncType<> 7 AND EncType <> 11 AND EncType <> 12
		THEN
			IF getValue(IDxGrp:= 16#5000,	IDxOffs := 16#101,	LEN := SIZEOF(_UINT),	pActValue := ADR(_UINT),  pSetValue := 0)
			THEN
				SetCalibrInvertDirForCamSearch :=CalibrInvertDirForCamSearch := TO_BOOL(_UINT);
				
			END_IF
		ELSE
			state											:= state +1;
		END_IF		
		
	1039: (* Calibration impuls direction inverted (of cam) *******************************************************)
		IF EncType <> 2 AND EncType <> 5 AND EncType<> 7 AND EncType <> 11 AND EncType <> 12
		THEN
			IF getValue(IDxGrp:= 16#5000,	IDxOffs := 16#102,	LEN := SIZEOF(_UINT),	pActValue := ADR(_UINT),  pSetValue := 0)
			THEN
				SetCalibrInvertDirForSyncImpSearch :=CalibrInvertDirForSyncImpSearch := TO_BOOL(_UINT);
				
			END_IF
	
		ELSE
			state											:= state +1;
		END_IF	
		
	1040: (* Calibration mode *******************************************************)
		IF EncType <> 2 AND EncType <> 5 AND EncType<> 7 AND EncType <> 11 AND EncType <> 12
		THEN
			getValue(IDxGrp:= 16#5000,	IDxOffs := 16#107,	LEN := SIZEOF(CalibrationMode),	pActValue := ADR(CalibrationMode),  pSetValue := ADR(SetCalibrationMode));
		ELSE
			state											:= state +1;
		END_IF
		
	1041: (* Scaling numerator **************************************)
		getValue(IDxGrp:= 16#5000,	IDxOffs := 16#23,	LEN := SIZEOF(EncScalingNumerator),	pActValue := ADR(EncScalingNumerator),  pSetValue := ADR(SetEncScalingNumerator) );	
			
	1042: (* Scaling denumerator **************************************)
		getValue(IDxGrp:= 16#5000,	IDxOffs := 16#24,	LEN := SIZEOF(EncScalingDenominator),	pActValue := ADR(EncScalingDenominator),  pSetValue := ADR(SetEncScalingDenominator) );	
		
	1043: (* Reference system **************************************)
		getValue(IDxGrp:= 16#5000,	IDxOffs := 16#19,	LEN := SIZEOF(ReferenceSystem),	pActValue := ADR(ReferenceSystem),  pSetValue := ADR(SetReferenceSystem) );	

	1044: (* Schleppabstand Filter Time ***********************************************************************)	
		getValue(IDxGrp:= 16#6000,	IDxOffs := 16#13,	LEN := SIZEOF(MaxPosLagFilterTime),	pActValue := ADR(MaxPosLagFilterTime),  pSetValue := ADR(SetMaxPosLagFilterTime) );

							
	ELSE
		state												:= 1;
	END_CASE

(*********************************************************************************************)
END_METHOD

METHOD PROTECTED seqWrite : BOOL //Return value = TRUE if execution finished 
VAR_IN_OUT
	State							:	INT;
END_VAR
(* Write axis parameter ********************************************************************)
	CASE state OF
	1..99: //Wite application spec parameter 
		seqWrite											:= TRUE;
		
	1001: (* Endlagenlimit pos.beschreiben ********************************************************)
		setValue(IDxGrp:= 16#5000,	IDxOffs := 16#E,	LEN := SIZEOF(SetLimitPos),		pActValue := ADR(LimitPos),		pSetValue := ADR(SetLimitPos));

	1002: (* Endlagenlimit neg.beschreiben ********************************************************)
		setValue(IDxGrp:= 16#5000,	IDxOffs := 16#D,	LEN := SIZEOF(SetLimitNeg),		pActValue := ADR(LimitNeg),		pSetValue := ADR(SetLimitNeg));

	1003: (* Endlagenlimit pos. aktiv ****************************************************************)
		IF NOT (SetLimitPosActive XOR LimitPosActive)
			AND NOT WriteAdsPara.BUSY
		THEN 
			state 											:= state + 1;
		ELSE
			_UINT											:= TO_UINT(SetLimitPosActive);
			LimitPosActive									:= SetLimitPosActive;
			setValue(IDxGrp:= 16#5000,	IDxOffs := 16#C,	LEN := SIZEOF(_UINT),		pActValue := 0,		pSetValue := ADR(_UINT));
		END_IF
		
	1004: (* Endlagenlimit neg.aktiv *****************************************************************)
		IF NOT (SetLimitNegActive XOR LimitNegActive) 
			AND NOT WriteAdsPara.BUSY
		THEN 
			state 											:= state + 1;
		ELSE
			_UINT											:= TO_UINT(SetLimitNegActive);
			LimitNegActive									:= SetLimitNegActive; 
			setValue(IDxGrp:= 16#5000,	IDxOffs := 16#B,	LEN := SIZEOF(_UINT),		pActValue := 0,		pSetValue := ADR(_UINT));
		END_IF

	1005: (* Zielfenster setzen **********************************************************************)
		setValue(IDxGrp:= 16#4000,	IDxOffs := 16#16,	LEN := SIZEOF(SetTargetPosWindow),		pActValue := ADR(TargetPosWindow),		pSetValue := ADR(SetTargetPosWindow));

	1006: (* Positionsfenster setzen *****************************************************************)
		setValue(IDxGrp:= 16#4000,	IDxOffs := 16#10,	LEN := SIZEOF(SetPosRangeWindow),		pActValue := ADR(PosRangeWindow),	pSetValue := ADR(SetPosRangeWindow));
		
	1007: (* Bezugsgeschwindigkeit setzen ********************************************************)
		IF AxisType = 2
		THEN 
			state 											:= state +1;
		ELSE
			setValue(IDxGrp:= 16#7000,	IDxOffs := 16#101,	LEN := SIZEOF(SetDynamicsRefVelocity),pActValue := ADR(DynamicsRefVelocity),	pSetValue := ADR(SetDynamicsRefVelocity));
		END_IF


	1008: (* Max.Geschwindigkeit setzen ************************************************************)
		IF AxisType = 2 
		THEN 
			state 											:= state +1;
		ELSE
			setValue(IDxGrp:= 16#4000,	IDxOffs := 16#27,	LEN := SIZEOF(SetDynamicsMaxVelocity),pActValue := ADR(DynamicsMaxVelocity),	pSetValue := ADR(SetDynamicsMaxVelocity));
		END_IF

	1009: (* G0 Geschwindigkeit setzen ****************************************************************)
		setValue(IDxGrp:= 16#4000,	IDxOffs := 16#A,	LEN := SIZEOF(SetG0Velocity),	pActValue := ADR(G0Velocity),	pSetValue := ADR(SetG0Velocity));

	1010: (* Ref.Geschwindigkeit fast setzen *******************************************************)
		setValue(IDxGrp:= 16#4000,	IDxOffs := 16#6,	LEN := SIZEOF(SetRefVelocityPos),	pActValue := ADR(RefVelocityPos),	pSetValue := ADR(SetRefVelocityPos));

	1011: (* Ref.Geschwindigkeit slow setzen *****************************************************)
		setValue(IDxGrp:= 16#4000,	IDxOffs := 16#7,	LEN := SIZEOF(SetRefVelocityNeg),	pActValue := ADR(RefVelocityNeg),	pSetValue := ADR(SetRefVelocityNeg));

	1012: (* Man.Geschwindigkeit fast setzen ******************************************************)
		setValue(IDxGrp:= 16#4000,	IDxOffs := 16#9,	LEN := SIZEOF(SetManVelocityFast),	pActValue := ADR(ManVelocityFast),	pSetValue := ADR(SetManVelocityFast));
		

	1013: (* Man.Geschwindigkeit slow setzen ******************************************************)
		setValue(IDxGrp:= 16#4000,	IDxOffs := 16#8,	LEN := SIZEOF(SetManVelocitySlow),	pActValue := ADR(ManVelocitySlow),	pSetValue := ADR(SetManVelocitySlow));

	1014: (* Kv setzen **************************************************************************************)
		IF AxisType = 2 
		THEN 
			state 											:= state +1;
		ELSE
			setValue(IDxGrp:= 16#6000,	IDxOffs := 16#102,	LEN := SIZEOF(SetKv),pActValue := ADR(Kv),	pSetValue := ADR(SetKv));
		END_IF

	1015: (* Ruck setzen ***********************************************************************************)
		IF AxisType = 2 
		THEN 
			state 											:= state +1;
		ELSE
			setValue(IDxGrp:= 16#4000,	IDxOffs := 16#103,	LEN := SIZEOF(SetJerk),pActValue := ADR(Jerk),	pSetValue := ADR(SetJerk));
		END_IF

	1016: (* Beschleunigung setzen **********************************************************************)
		IF AxisType = 2 
		THEN 
			state 											:= state +1;
		ELSE
			setValue(IDxGrp:= 16#4000,	IDxOffs := 16#101,	LEN := SIZEOF(SetAcc), pActValue := ADR(Acc),	pSetValue := ADR(SetAcc));
		END_IF
	
	1017: (* Verzoegerung setzen ************************************************************************)
		IF AxisType = 2 
		THEN 
			state 											:= state +1;
		ELSE
			setValue(IDxGrp:= 16#4000,	IDxOffs := 16#102,	LEN := SIZEOF(SetDec), pActValue := ADR(Dec),	pSetValue := ADR(SetDec));
		END_IF
		
	1018: (* Schleppabstand setzen **********************************************************************)
		setValue(IDxGrp:= 16#6000,	IDxOffs := 16#12,	LEN := SIZEOF(SetMaxPosLagValue),	pActValue := ADR(MaxPosLagValue),	pSetValue := ADR(SetMaxPosLagValue));

	1019: (* Reserverd *****************************************************************************)
		// Set scaling replaced by Num and Denum  setValue(IDxGrp:= 16#5000,	IDxOffs := 16#6,	LEN := SIZEOF(SetEncScaling),	pActValue := ADR(EncScaling),	pSetValue := ADR(SetEncScaling));
		state 												:= state +1 ;
		
	1020: (* Positions Offset setzen ****************************************************************)
		setValue(IDxGrp:= 16#5000,	IDxOffs := 16#7,	LEN := SIZEOF(SetPosBias),	pActValue := ADR(PosBias),	pSetValue := ADR(SetPosBias));
		
	1021: (* Referenzposition setzen ***************************************************************)
		IF EncType <> 2  AND EncType <> 5 AND EncType <> 7 AND EncType <> 11  AND EncType <> 12 
		THEN
			setValue(IDxGrp:= 16#5000,	IDxOffs := 16#103,	LEN := SIZEOF(SetCalibrationValue),	pActValue := ADR(CalibrationValue),	pSetValue := ADR(SetCalibrationValue));
		ELSE
			state 											:= state +1 ;
		END_IF

	1022: (* Bremsweg positiv **********************************************************************)
		IF AxisType = 2 
		THEN 
			state 											:= state +1;
		ELSE
			setValue(IDxGrp:= 16#4000,	IDxOffs := 16#303,	LEN := SIZEOF(SetBreakingDistancePos), pActValue := ADR(BreakingDistancePos),	pSetValue := ADR(SetBreakingDistancePos));
		END_IF

	1023: (* Bremsweg negativ *********************************************************************)
		IF AxisType = 2
		THEN 
			state 											:= state +1;
		ELSE
			setValue(IDxGrp:= 16#4000,	IDxOffs := 16#304,	LEN := SIZEOF(SetBreakingDistanceNeg), pActValue := ADR(BreakingDistanceNeg),	pSetValue := ADR(SetBreakingDistanceNeg));
		END_IF

	1024: (* Schleppueberwachung ****************************************************************************)
		IF SetMaxPosLagMonitoring = MaxPosLagMonitoring AND NOT WriteAdsPara.BUSY
		THEN 
			state 											:= state +1;
		ELSE
			_UINT											:= TO_UINT(SetMaxPosLagMonitoring);
			MaxPosLagMonitoring								:= SetMaxPosLagMonitoring;					
			setValue(IDxGrp:= 16#6000,	IDxOffs := 16#10,	LEN := SIZEOF(_UINT),	pActValue := 0,	pSetValue := ADR(_UINT));
		END_IF

	1025: (* Referenzierflag ****************************************************************************)
		IF RefFlag = SetRefFlag AND NOT WriteAdsPara.BUSY
		THEN 
			state 											:= state +1;
		ELSE
			_UINT											:= TO_UINT(SetRefFlag);
			RefFlag											:= SetRefFlag;
			setValue(IDxGrp:= 16#5100,	IDxOffs := 16#9,	LEN := SIZEOF(_UINT), pActValue := 0,	pSetValue := ADR(_UINT));
		END_IF
		
	1026: (* PosfensterAktiv ****************************************************************************)
		IF SetPosRangeWindowMonitoring = PosRangeWindowMonitoring AND NOT WriteAdsPara.BUSY
		THEN 
			state 											:= state +1;
		ELSE
			_UINT											:= TO_UINT(SetPosRangeWindowMonitoring);
			PosRangeWindowMonitoring						:= SetPosRangeWindowMonitoring;
			setValue(IDxGrp:= 16#4000,	IDxOffs := 16#F,	LEN := SIZEOF(_UINT), pActValue := 0,	pSetValue := ADR(_UINT));
		END_IF

	1027: (* ZielfensterAktiv ****************************************************************************)
		IF SetTargetPosWindowMonitoring = TargetPosWindowMonitoring AND NOT WriteAdsPara.BUSY
		THEN 
			state 											:= state +1;
		ELSE
			_UINT											:= TO_UINT(SetTargetPosWindowMonitoring);
			TargetPosWindowMonitoring						:= SetTargetPosWindowMonitoring;
			setValue(IDxGrp:= 16#4000,	IDxOffs := 16#15,	LEN := SIZEOF(_UINT), pActValue := 0,	pSetValue := ADR(_UINT));
		END_IF

	1028: (* Modulofaktor ****************************************************************************)
		setValue(IDxGrp:= 16#5000,	IDxOffs := 16#9,	LEN := SIZEOF(SetModuloFactor), pActValue := ADR(ModuloFactor),	pSetValue := ADR(SetModuloFactor));
		
	1029: (* Enc. Zaehlrichtung ****************************************************************************)
		IF SetInvertEncCoutingDir = InvertEncCoutingDir AND NOT WriteAdsPara.BUSY
		THEN 
			state 											:= state +1;
		ELSE
			_UINT											:= TO_UINT(SetInvertEncCoutingDir);
			InvertEncCoutingDir								:= SetInvertEncCoutingDir;
			setValue(IDxGrp:= 16#5000,	IDxOffs := 16#8,	LEN := SIZEOF(_UINT), pActValue := 0,	pSetValue := ADR(_UINT));
		END_IF

	1030: (* Drive  ****************************************************************************)
		IF SetInvertMotorPolarity = InvertMotorPolarity AND NOT WriteAdsPara.BUSY
		THEN 
			state 											:= state +1;
		ELSE
			_UINT											:= TO_UINT(SetInvertMotorPolarity);
			InvertMotorPolarity								:= SetInvertMotorPolarity;
			setValue(IDxGrp:= 16#7000,	IDxOffs := 16#6,	LEN := SIZEOF(_UINT), pActValue := 0,	pSetValue := ADR(_UINT));
		END_IF
		
		
	1031: (* Enc. Modulo start tolerance ****************************************************************************)
		setValue(IDxGrp:= 16#5000,	IDxOffs := 16#1B,	LEN := SIZEOF(SetToleranceWindowModuloStart), pActValue := ADR(ToleranceWindowModuloStart),	pSetValue := ADR(SetToleranceWindowModuloStart));

	1032: (* Set calibration cam search direction inverted ***************************************************************)
		IF SetCalibrInvertDirForCamSearch <> CalibrInvertDirForCamSearch 
			AND_THEN EncType <> 2  AND EncType <> 5 AND EncType <> 7 AND EncType <> 11  AND EncType <> 12
			AND NOT WriteAdsPara.BUSY
		THEN 
			state 											:= state +1;
		ELSE
			_UINT											:= TO_UINT(SetCalibrInvertDirForCamSearch);
			CalibrInvertDirForCamSearch						:= SetCalibrInvertDirForCamSearch;
			setValue(IDxGrp:= 16#5000,	IDxOffs := 16#101,	LEN := SIZEOF(_UINT), pActValue := 0,	pSetValue := ADR(_UINT));
		END_IF

	1033: (* Set calibration impuls search direction inverted ***************************************************************)
		IF SetCalibrInvertDirForSyncImpSearch <> CalibrInvertDirForSyncImpSearch 
			AND_THEN EncType <> 2  AND EncType <> 5 AND EncType <> 7 AND EncType <> 11  AND EncType <> 12
			AND NOT WriteAdsPara.BUSY
		THEN 
			state 											:= state +1;
		ELSE
			_UINT											:= TO_UINT(SetCalibrInvertDirForSyncImpSearch);
			CalibrInvertDirForSyncImpSearch					:= SetCalibrInvertDirForSyncImpSearch;
			setValue(IDxGrp:= 16#5000,	IDxOffs := 16#102,	LEN := SIZEOF(_UINT), pActValue := 0,	pSetValue := ADR(_UINT));
		END_IF
		
	1034: (* Set calibration mode ***************************************************************)
		IF SetCalibrationMode <> CalibrationMode 
			AND_THEN EncType <> 2  AND EncType <> 5 AND EncType <> 7 AND EncType <> 11  AND EncType <> 12
			AND NOT WriteAdsPara.BUSY
		THEN 
			state 											:= state +1;		
		ELSE
			setValue(IDxGrp:= 16#5000,	IDxOffs := 16#107,	LEN := SIZEOF(SetCalibrationMode), pActValue := ADR(CalibrationMode),	pSetValue := ADR(SetCalibrationMode));
		END_IF

	1035: (* Scaling numerator **************************************)
		setValue(IDxGrp:= 16#5000,	IDxOffs := 16#23,	LEN := SIZEOF(SetEncScalingNumerator),	pActValue := ADR(EncScalingNumerator),  pSetValue := ADR(SetEncScalingNumerator) );	
			
	1036: (* Scaling denumerator **************************************)
		setValue(IDxGrp:= 16#5000,	IDxOffs := 16#24,	LEN := SIZEOF(SetEncScalingDenominator),	pActValue := ADR(EncScalingDenominator),  pSetValue := ADR(SetEncScalingDenominator) );
		
		//Calculate Act Scaling 
		IF NOT Error THEN  EncScaling	:= EncScalingNumerator / EncScalingDenominator; END_IF
		
	1037: (* Reference system **************************************)
		setValue(IDxGrp:= 16#5000,	IDxOffs := 16#19,	LEN := SIZEOF(SetReferenceSystem),	pActValue := ADR(ReferenceSystem),  pSetValue := ADR(SetReferenceSystem) );	
	
	1038: (* Schleppueberwachung Zeit ****************************************************************************)
		setValue(IDxGrp:= 16#6000,	IDxOffs := 16#13,	LEN := SIZEOF(SetMaxPosLagFilterTime),	pActValue := ADR(MaxPosLagFilterTime),	pSetValue := ADR(SetMaxPosLagFilterTime));
	
	ELSE
		state 												:= 1 ;
	END_CASE
	
(***********************************************************************************************)
END_METHOD

METHOD PROTECTED setValue : BOOL //Return value = TRUE if execution finished and state incremented 
VAR_INPUT
	IDxGrp						:	UDINT;
	IDxOffs						:	UDINT;
	Len							:	UDINT;
	pActValue					:	PVOID; //Address of variable for actual value, can be zero if no corresponding acual value variable exists
	pSetValue					:	PVOID; //Address of variable for set value variable
END_VAR

IF pActValue <> 0 AND pSetValue <> 0 AND_THEN MEMCMP(pSetValue, pActValue, Len) = 0
THEN //Skip write parameter if set and actual value are equel
	state													:= state + 1;	
	setValue												:= TRUE;
ELSE
	WriteAdsPara( Write := TRUE, IdxGrp :=IDxGrp+AxisId, IdxOffs:=IDxOffs, LEN:=Len, SrcAddr:=pSetValue );
	IF NOT WriteAdsPara.BUSY
	THEN
		IF NOT WriteAdsPara.ERR
		THEN
			IF pActValue <> 0 THEN MEMCPY(pActValue, pSetValue, Len); END_IF	
			state											:= state + 1;
		ELSE
			Busy											:= FALSE;
			Error											:= TRUE;
			ErrorId											:= WriteAdsPara.ERRID;
			ErrorText										:= CONCAT('Error write parameter in state:' , TO_STRING(state * -1));
			ErrorText										:= CONCAT(ErrorText , ' Id:');
			ErrorText										:= CONCAT(ErrorText , TO_STRING(ErrorId));
			State											:= 9999;
		END_IF
		WriteAdsPara (Write := FALSE);
		setValue											:= TRUE;
	END_IF		
END_IF
END_METHOD

END_FUNCTION_BLOCK

// POUs/Motion/TF50xx-NC/00_Base/I_AxNcPTP
INTERFACE I_AxNcPTP EXTENDS I_AxNcBase

{attribute 'monitoring' := 'call'}
PROPERTY rMotion : REFERENCE TO AxMotion
GET
END_GET
END_PROPERTY

END_INTERFACE

// POUs/Motion/TF50xx-NC/01_Main/AxMotion
{attribute 'no_check'}
//Nc-axis motion control - start/stop axis  
//based on Tc2_MC2 library
FUNCTION_BLOCK AxMotion EXTENDS AxFbBase
VAR_OUTPUT CONSTANT
	FNC_HALT												:	INT := 0;
	FNC_STOP												:	INT := 1;
	FNC_MOVE_JOG											:	INT := 2;
	FNC_MOVE_ABS											:	INT := 3;
	FNC_MOVE_REL											:	INT := 4;
	FNC_MOVE_ADD											:	INT := 5;
	FNC_MOVE_MOD											:	INT := 6;
	FNC_MOVE_VELO											:	INT := 7;
END_VAR
VAR_INPUT
	Fnc														:	INT (FNC_HALT..FNC_MOVE_VELO) := FNC_HALT;
	JogFwd													:	BOOL := FALSE;
	JogBwd													:	BOOL	:= FALSE;
	BufferMode												:	MC_BufferMode := MC_Aborting;(* 	MC_Aborting,
																											MC_Buffered,
																											MC_BlendingLow,
																											MC_BlendingPrevious,
																											MC_BlendingNext,
																											MC_BlendingHigh *)
	Direction												:	MC_Direction := MC_POSITIVE_DIRECTION;	(*	MC_POSITIVE_DIRECTION,
																														   MC_SHORTeSTATE.WAY,
																														   MC_NEGATIVE_DIRECTION,
																														   MC_CURRENT_DIRECTION *)
	JogMode													:	E_JogMode := MC_JOGMODE_STANDARD_SLOW;	(*	MC_JOGMODE_STANDARD_SLOW
																															MC_JOGMODE_STANDARD_FAST
																															MC_JOGMODE_CONTINOUS
																															MC_JOGMODE_INCHING 
																															MC_JOGeMODE.INCHING_MODULO *)
	Target													:	LREAL; (* Zielposition *)
	Velo														: 	LREAL; (* Zielgeschwindigkeit *)
	Jerk														:	LREAL := 0.0 ; (* Bei 0 werden wird der Ruck aus dem TCManager uebernommen *)
	Acc														:	LREAL := 0.0; (* Bei 0 werden wird die Beschleunigung aus dem TCManager uebernommen *)
	Dec														:	LREAL := 0.0; (* Bei 0 werden wird die Verzoegerung aus dem TCManager uebernommen *)
	MoveOptions												:	ST_MoveOptions;
END_VAR                     								
VAR_IN_OUT                  								
END_VAR                     								
VAR_OUTPUT                  								
END_VAR
VAR
(* Zwischenspeicher **************************************************************************)
	MemFnc													:	INT := -1;
	MemFncAct												:	INT := -1;
	MCFctTxt												:	STRING(25);
	TrigID													:	INT := 2; (* um mit Trig 1 zu starten *)
	MemBufferMode											:	MC_BufferMode;
	ActSetTarget											:	LREAL;
	ActSetVelo												:	LREAL;
	BusyIntern												:	BOOL;

(* Timer *)

(* Trigger *)
	rtExecuteMethod											:	R_TRIG;

(* Instanzierung der MC Bausteine *******************************************************)
	MC_Halt													: 	MC_Halt;
	MC_Stop													: 	MC_Stop;
	MC_MoveVeloPreTrig										: 	MC_MoveVelocity;
	MC_Jog													: 	MC_Jog;

(* Durch entfernen der Kommentarsymbole koennen noch weitere benötigte MC_Move Varianten
	mit ins Programm genommen werden 
*)
	MC_MoveAbsolute											: 	ARRAY[1..2] OF MC_MoveAbsolute;
	MC_MoveModulo											: 	ARRAY[1..2] OF MC_MoveModulo;
	MC_MoveRelative											: 	ARRAY[1..2] OF MC_MoveRelative;
	MC_MoveAdditive											: 	ARRAY[1..2] OF MC_MoveAdditive; 
	MC_MoveVelocity											: 	ARRAY[1..2] OF MC_MoveVelocity; 

(* Dummy Speicher **********************************************************)
	i														: INT := 0 ;

(* Skalierungsfaktor ermitteln *********************************************
	Skalierungsfaktor von 0.1 eintragen. Istpositon "Anfang" merken.
	Antrieb um einen realen Wert "X" mm verfahren. Differenz der
	momentanen Istposition zur Istposition "Anfang" ermitteln.
	SKalierungsfaktor =		realer Fahrweg 
							---------------------------
							Differenz der Istpositionen
*)
END_VAR

	(* Axis motion control 													*)
	(************************************************************************)

